LIN {X 0,Y 355.235,Z 349.049,A -85,B 0,C 180,E1 -13317.733,E2 -13317.733} C_VEL
LIN {X 0,Y 355.386,Z 349.032,A -85,B 0,C 180,E1 -13320.001,E2 -13320.001} C_VEL
LIN {X 0,Y 355.236,Z 349.048,A -85,B 0,C 180,E1 -13322.269,E2 -13322.269} C_VEL
LIN {X 0,Y 355.128,Z 349.059,A -85,B 0,C 180,E1 -13326.82,E2 -13326.82} C_VEL
LIN {X 0,Y 355.007,Z 349.075,A -85,B 0,C 180,E1 -13329.114,E2 -13329.114} C_VEL
LIN {X 0,Y 354.917,Z 349.085,A -85,B 0,C 180,E1 -13332.582,E2 -13332.582} C_VEL
LIN {X 0,Y 354.88,Z 349.091,A -85,B 0,C 180,E1 -13336.097,E2 -13336.097} C_VEL
LIN {X 0,Y 354.892,Z 349.088,A -85,B 0,C 180,E1 -13338.474,E2 -13338.474} C_VEL
LIN {X 0,Y 354.826,Z 349.097,A -85,B 0,C 180,E1 -13342.108,E2 -13342.108} C_VEL
LIN {X 0,Y 354.891,Z 349.09,A -85,B 0,C 180,E1 -13345.829,E2 -13345.829} C_VEL
LIN {X 0,Y 354.847,Z 349.096,A -85,B 0,C 180,E1 -13349.68,E2 -13349.68} C_VEL
LIN {X 0,Y 354.799,Z 349.101,A -85,B 0,C 180,E1 -13353.704,E2 -13353.704} C_VEL
LIN {X 0,Y 354.792,Z 349.102,A -85,B 0,C 180,E1 -13356.461,E2 -13356.461} C_VEL
LIN {X 0,Y 354.818,Z 349.099,A -85,B 0,C 180,E1 -13359.425,E2 -13359.425} C_VEL
LIN {X 0,Y 354.783,Z 349.107,A -85,B 0,C 180,E1 -13362.869,E2 -13362.869} C_VEL
LIN {X 0,Y 354.771,Z 349.104,A -85,B 0,C 180,E1 -13366.107,E2 -13366.107} C_VEL
LIN {X 0,Y 354.897,Z 349.091,A -85,B 0,C 180,E1 -13370.299,E2 -13370.299} C_VEL
LIN {X 0,Y 354.925,Z 349.475,A -85,B 0,C 180,E1 -13370.683,E2 -13370.683} C_VEL
LIN {X 0,Y 355.893,Z 355.008,A -85,B 0,C 180,E1 -13374.062,E2 -13374.062} C_VEL
LIN {X 0,Y 356.377,Z 359.185,A -85,B 0,C 180,E1 -13376.485,E2 -13376.485} C_VEL
LIN {X 0,Y 356.221,Z 361.976,A -85,B 0,C 180,E1 -13378.035,E2 -13378.035} C_VEL
LIN {X 0,Y 355.439,Z 368.762,A -85,B 0,C 180,E1 -13381.672,E2 -13381.672} C_VEL
LIN {X 0,Y 354.767,Z 375.912,A -85,B 0,C 180,E1 -13385.419,E2 -13385.419} C_VEL
LIN {X 0,Y 354.249,Z 383.077,A -85,B 0,C 180,E1 -13389.079,E2 -13389.079} C_VEL
LIN {X 0,Y 353.744,Z 391.414,A -85,B 0,C 180,E1 -13393.259,E2 -13393.259} C_VEL
LIN {X 0,Y 353.648,Z 393.722,A -85,B 0,C 180,E1 -13394.347,E2 -13394.347} C_VEL
LIN {X 0,Y 355.033,Z 405.955,A -85,B 0,C 180,E1 -13394.943,E2 -13394.943} C_VEL
LIN {X 0,Y 355.952,Z 415.878,A -85,B 0,C 180,E1 -13395.628,E2 -13395.628} C_VEL
LIN {X 0,Y 356.321,Z 423.872,A -85,B 0,C 180,E1 -13396.311,E2 -13396.311} C_VEL
LIN {X 0,Y 356.015,Z 430.965,A -85,B 0,C 180,E1 -13397.025,E2 -13397.025} C_VEL
LIN {X 0,Y 355.341,Z 439.04,A -85,B 0,C 180,E1 -13398.016,E2 -13398.016} C_VEL
LIN {X 0,Y 354.883,Z 444.875,A -85,B 0,C 180,E1 -13398.869,E2 -13398.869} C_VEL
LIN {X 0,Y 354.341,Z 451.371,A -85,B 0,C 180,E1 -13400.007,E2 -13400.007} C_VEL
LIN {X 0,Y 353.972,Z 456.779,A -85,B 0,C 180,E1 -13401.15,E2 -13401.15} C_VEL
LIN {X 0,Y 353.626,Z 462.253,A -85,B 0,C 180,E1 -13402.579,E2 -13402.579} C_VEL
LIN {X 0,Y 353.352,Z 466.492,A -85,B 0,C 180,E1 -13403.978,E2 -13403.978} C_VEL
LIN {X 0,Y 353.355,Z 469.884,A -85,B 0,C 180,E1 -13405.438,E2 -13405.438} C_VEL
LIN {X 0,Y 353.281,Z 471.864,A -85,B 0,C 180,E1 -13406.58,E2 -13406.58} C_VEL
LIN {X 0,Y 353.296,Z 473.328,A -85,B 0,C 180,E1 -13407.721,E2 -13407.721} C_VEL
LIN {X 0,Y 353.362,Z 474.262,A -85,B 0,C 180,E1 -13408.862,E2 -13408.862} C_VEL
LIN {X 0,Y 353.395,Z 474.597,A -85,B 0,C 180,E1 -13410.001,E2 -13410.001} C_VEL
LIN {X 0,Y 353.356,Z 474.442,A -85,B 0,C 180,E1 -13411.141,E2 -13411.141} C_VEL
LIN {X 0,Y 353.261,Z 473.814,A -85,B 0,C 180,E1 -13412.282,E2 -13412.282} C_VEL
LIN {X 0,Y 353.272,Z 472.711,A -85,B 0,C 180,E1 -13413.423,E2 -13413.423} C_VEL
LIN {X 0,Y 353.325,Z 469.93,A -85,B 0,C 180,E1 -13415.137,E2 -13415.137} C_VEL
LIN {X 0,Y 353.412,Z 467.446,A -85,B 0,C 180,E1 -13416.28,E2 -13416.28} C_VEL
LIN {X 0,Y 353.649,Z 464.318,A -85,B 0,C 180,E1 -13417.423,E2 -13417.423} C_VEL
LIN {X 0,Y 354.118,Z 458.219,A -85,B 0,C 180,E1 -13419.137,E2 -13419.137} C_VEL
LIN {X 0,Y 354.581,Z 453.195,A -85,B 0,C 180,E1 -13420.277,E2 -13420.277} C_VEL
LIN {X 0,Y 355.196,Z 447.164,A -85,B 0,C 180,E1 -13421.413,E2 -13421.413} C_VEL
LIN {X 0,Y 355.86,Z 439.855,A -85,B 0,C 180,E1 -13422.549,E2 -13422.549} C_VEL
LIN {X 0,Y 356.656,Z 432.1,A -85,B 0,C 180,E1 -13423.534,E2 -13423.534} C_VEL
LIN {X 0,Y 357.137,Z 425.476,A -85,B 0,C 180,E1 -13424.241,E2 -13424.241} C_VEL
LIN {X 0,Y 356.862,Z 416.272,A -85,B 0,C 180,E1 -13425.081,E2 -13425.081} C_VEL
LIN {X 0,Y 356.041,Z 407.363,A -85,B 0,C 180,E1 -13425.75,E2 -13425.75} C_VEL
LIN {X 0,Y 354.507,Z 396.758,A -85,B 0,C 180,E1 -13426.388,E2 -13426.388} C_VEL
LIN {X 0,Y 353.78,Z 392.415,A -85,B 0,C 180,E1 -13426.594,E2 -13426.594} C_VEL
LIN {X 0,Y 354.187,Z 385.023,A -85,B 0,C 180,E1 -13430.32,E2 -13430.32} C_VEL
LIN {X 0,Y 354.791,Z 377.309,A -85,B 0,C 180,E1 -13434.326,E2 -13434.326} C_VEL
LIN {X 0,Y 355.443,Z 371.062,A -85,B 0,C 180,E1 -13437.689,E2 -13437.689} C_VEL
LIN {X 0,Y 356.313,Z 364.375,A -85,B 0,C 180,E1 -13441.442,E2 -13441.442} C_VEL
LIN {X 0,Y 356.63,Z 360.91,A -85,B 0,C 180,E1 -13443.491,E2 -13443.491} C_VEL
LIN {X 0,Y 356.164,Z 356.993,A -85,B 0,C 180,E1 -13445.998,E2 -13445.998} C_VEL
LIN {X 0,Y 355.369,Z 351.925,A -85,B 0,C 180,E1 -13449.529,E2 -13449.529} C_VEL
LIN {X 0,Y 354.824,Z 349.11,A -85,B 0,C 180,E1 -13451.712,E2 -13451.712} C_VEL
LIN {X 0,Y 354.771,Z 349.112,A -85,B 0,C 180,E1 -13455.494,E2 -13455.494} C_VEL
LIN {X 0,Y 354.795,Z 349.105,A -85,B 0,C 180,E1 -13459.179,E2 -13459.179} C_VEL
LIN {X 0,Y 354.814,Z 349.102,A -85,B 0,C 180,E1 -13462.403,E2 -13462.403} C_VEL
LIN {X 0,Y 354.819,Z 349.102,A -85,B 0,C 180,E1 -13464.941,E2 -13464.941} C_VEL
LIN {X 0,Y 354.801,Z 349.103,A -85,B 0,C 180,E1 -13468.405,E2 -13468.405} C_VEL
LIN {X 0,Y 354.854,Z 349.097,A -85,B 0,C 180,E1 -13471.618,E2 -13471.618} C_VEL
LIN {X 0,Y 354.907,Z 349.091,A -85,B 0,C 180,E1 -13474.172,E2 -13474.172} C_VEL
LIN {X 0,Y 354.843,Z 349.098,A -85,B 0,C 180,E1 -13477.894,E2 -13477.894} C_VEL
LIN {X 0,Y 354.93,Z 349.087,A -85,B 0,C 180,E1 -13481.891,E2 -13481.891} C_VEL
LIN {X 0,Y 354.95,Z 349.085,A -85,B 0,C 180,E1 -13485.981,E2 -13485.981} C_VEL
LIN {X 0,Y 354.963,Z 349.084,A -85,B 0,C 180,E1 -13489.734,E2 -13489.734} C_VEL
LIN {X 0,Y 355.106,Z 349.065,A -85,B 0,C 180,E1 -13493.179,E2 -13493.179} C_VEL
LIN {X 0,Y 355.246,Z 349.048,A -85,B 0,C 180,E1 -13497.731,E2 -13497.731} C_VEL
LIN {X 0,Y 355.381,Z 349.033,A -85,B 0,C 180,E1 -13499.999,E2 -13499.999} C_VEL
LIN {X 0,Y 355.248,Z 349.048,A -85,B 0,C 180,E1 -13502.266,E2 -13502.266} C_VEL
LIN {X 0,Y 355.117,Z 349.065,A -85,B 0,C 180,E1 -13506.818,E2 -13506.818} C_VEL
LIN {X 0,Y 354.96,Z 349.084,A -85,B 0,C 180,E1 -13510.263,E2 -13510.263} C_VEL
LIN {X 0,Y 354.943,Z 349.089,A -85,B 0,C 180,E1 -13514.015,E2 -13514.015} C_VEL
LIN {X 0,Y 354.751,Z 349.114,A -85,B 0,C 180,E1 -13517.286,E2 -13517.286} C_VEL
LIN {X 0,Y 354.61,Z 349.14,A -85,B 0,C 180,E1 -13518.486,E2 -13518.486} C_VEL
LIN {X 0,Y 354.486,Z 351.743,A -85,B 0,C 180,E1 -13521.278,E2 -13521.278} C_VEL
LIN {X 0,Y 354.24,Z 354.97,A -85,B 0,C 180,E1 -13524.621,E2 -13524.621} C_VEL
LIN {X 0,Y 354.088,Z 357.477,A -85,B 0,C 180,E1 -13527.16,E2 -13527.16} C_VEL
LIN {X 0,Y 353.925,Z 360.115,A -85,B 0,C 180,E1 -13529.763,E2 -13529.763} C_VEL
LIN {X 0,Y 353.767,Z 363.986,A -85,B 0,C 180,E1 -13533.509,E2 -13533.509} C_VEL
LIN {X 0,Y 356.374,Z 374.506,A -85,B 0,C 180,E1 -13534.195,E2 -13534.195} C_VEL
LIN {X 0,Y 358.039,Z 383.016,A -85,B 0,C 180,E1 -13534.867,E2 -13534.867} C_VEL
LIN {X 0,Y 358.578,Z 389.237,A -85,B 0,C 180,E1 -13535.407,E2 -13535.407} C_VEL
LIN {X 0,Y 357.779,Z 399.313,A -85,B 0,C 180,E1 -13536.426,E2 -13536.426} C_VEL
LIN {X 0,Y 357.04,Z 406.286,A -85,B 0,C 180,E1 -13537.29,E2 -13537.29} C_VEL
LIN {X 0,Y 356.525,Z 412.401,A -85,B 0,C 180,E1 -13538.2,E2 -13538.2} C_VEL
LIN {X 0,Y 355.812,Z 419.035,A -85,B 0,C 180,E1 -13539.391,E2 -13539.391} C_VEL
LIN {X 0,Y 355.266,Z 423.977,A -85,B 0,C 180,E1 -13540.454,E2 -13540.454} C_VEL
LIN {X 0,Y 354.667,Z 429.227,A -85,B 0,C 180,E1 -13541.838,E2 -13541.838} C_VEL
LIN {X 0,Y 354.332,Z 432.253,A -85,B 0,C 180,E1 -13542.786,E2 -13542.786} C_VEL
LIN {X 0,Y 353.898,Z 436.127,A -85,B 0,C 180,E1 -13544.362,E2 -13544.362} C_VEL
LIN {X 0,Y 353.594,Z 438.873,A -85,B 0,C 180,E1 -13545.919,E2 -13545.919} C_VEL
LIN {X 0,Y 353.3,Z 440.605,A -85,B 0,C 180,E1 -13547.44,E2 -13547.44} C_VEL
LIN {X 0,Y 353.163,Z 441.468,A -85,B 0,C 180,E1 -13549.128,E2 -13549.128} C_VEL
LIN {X 0,Y 353.164,Z 441.225,A -85,B 0,C 180,E1 -13550.903,E2 -13550.903} C_VEL
LIN {X 0,Y 353.286,Z 439.695,A -85,B 0,C 180,E1 -13552.721,E2 -13552.721} C_VEL
LIN {X 0,Y 353.468,Z 437.782,A -85,B 0,C 180,E1 -13554.02,E2 -13554.02} C_VEL
LIN {X 0,Y 353.702,Z 434.686,A -85,B 0,C 180,E1 -13555.507,E2 -13555.507} C_VEL
LIN {X 0,Y 354.067,Z 430.281,A -85,B 0,C 180,E1 -13557.061,E2 -13557.061} C_VEL
LIN {X 0,Y 354.468,Z 425.095,A -85,B 0,C 180,E1 -13558.488,E2 -13558.488} C_VEL
LIN {X 0,Y 354.94,Z 419.788,A -85,B 0,C 180,E1 -13559.673,E2 -13559.673} C_VEL
LIN {X 0,Y 355.448,Z 413.918,A -85,B 0,C 180,E1 -13560.762,E2 -13560.762} C_VEL
LIN {X 0,Y 355.894,Z 407.866,A -85,B 0,C 180,E1 -13561.708,E2 -13561.708} C_VEL
LIN {X 0,Y 356.453,Z 400.719,A -85,B 0,C 180,E1 -13562.641,E2 -13562.641} C_VEL
LIN {X 0,Y 357.061,Z 392.116,A -85,B 0,C 180,E1 -13563.555,E2 -13563.555} C_VEL
LIN {X 0,Y 357.398,Z 384.562,A -85,B 0,C 180,E1 -13564.209,E2 -13564.209} C_VEL
LIN {X 0,Y 356.037,Z 375.647,A -85,B 0,C 180,E1 -13564.886,E2 -13564.886} C_VEL
LIN {X 0,Y 354.144,Z 365.686,A -85,B 0,C 180,E1 -13565.481,E2 -13565.481} C_VEL
LIN {X 0,Y 353.599,Z 362.774,A -85,B 0,C 180,E1 -13565.663,E2 -13565.663} C_VEL
LIN {X 0,Y 353.651,Z 358.953,A -85,B 0,C 180,E1 -13569.065,E2 -13569.065} C_VEL
LIN {X 0,Y 353.885,Z 354.967,A -85,B 0,C 180,E1 -13572.668,E2 -13572.668} C_VEL
LIN {X 0,Y 354.106,Z 350.778,A -85,B 0,C 180,E1 -13576.527,E2 -13576.527} C_VEL
LIN {X 0,Y 354.133,Z 349.869,A -85,B 0,C 180,E1 -13577.389,E2 -13577.389} C_VEL
LIN {X 0,Y 354.239,Z 349.175,A -85,B 0,C 180,E1 -13578.555,E2 -13578.555} C_VEL
LIN {X 0,Y 354.905,Z 349.09,A -85,B 0,C 180,E1 -13582.031,E2 -13582.031} C_VEL
LIN {X 0,Y 355.06,Z 349.072,A -85,B 0,C 180,E1 -13584.319,E2 -13584.319} C_VEL
LIN {X 0,Y 355.236,Z 349.047,A -85,B 0,C 180,E1 -13587.731,E2 -13587.731} C_VEL
LIN {X 0,Y 355.387,Z 349.031,A -85,B 0,C 180,E1 -13589.999,E2 -13589.999} C_VEL
LIN {X 0,Y 355.236,Z 349.049,A -85,B 0,C 180,E1 -13592.266,E2 -13592.266} C_VEL
LIN {X 0,Y 355.131,Z 349.059,A -85,B 0,C 180,E1 -13596.818,E2 -13596.818} C_VEL
LIN {X 0,Y 355.005,Z 349.074,A -85,B 0,C 180,E1 -13599.111,E2 -13599.111} C_VEL
LIN {X 0,Y 354.914,Z 349.086,A -85,B 0,C 180,E1 -13602.579,E2 -13602.579} C_VEL
LIN {X 0,Y 354.877,Z 349.093,A -85,B 0,C 180,E1 -13606.095,E2 -13606.095} C_VEL
LIN {X 0,Y 354.888,Z 349.089,A -85,B 0,C 180,E1 -13608.471,E2 -13608.471} C_VEL
LIN {X 0,Y 354.821,Z 349.099,A -85,B 0,C 180,E1 -13612.105,E2 -13612.105} C_VEL
LIN {X 0,Y 354.886,Z 349.092,A -85,B 0,C 180,E1 -13615.827,E2 -13615.827} C_VEL
LIN {X 0,Y 354.84,Z 349.098,A -85,B 0,C 180,E1 -13619.678,E2 -13619.678} C_VEL
LIN {X 0,Y 354.792,Z 349.103,A -85,B 0,C 180,E1 -13623.701,E2 -13623.701} C_VEL
LIN {X 0,Y 354.789,Z 349.101,A -85,B 0,C 180,E1 -13626.458,E2 -13626.458} C_VEL
LIN {X 0,Y 354.811,Z 349.102,A -85,B 0,C 180,E1 -13629.424,E2 -13629.424} C_VEL
LIN {X 0,Y 354.827,Z 349.1,A -85,B 0,C 180,E1 -13632.876,E2 -13632.876} C_VEL
LIN {X 0,Y 354.853,Z 349.093,A -85,B 0,C 180,E1 -13634.072,E2 -13634.072} C_VEL
LIN {X 0,Y 354.196,Z 349.18,A -85,B 0,C 180,E1 -13635.018,E2 -13635.018} C_VEL
LIN {X 0,Y 351.315,Z 349.536,A -85,B 0,C 180,E1 -13636.556,E2 -13636.556} C_VEL
LIN {X 0,Y 348.871,Z 349.838,A -85,B 0,C 180,E1 -13637.801,E2 -13637.801} C_VEL
LIN {X 0,Y 347.831,Z 349.972,A -85,B 0,C 180,E1 -13638.765,E2 -13638.765} C_VEL
LIN {X 0,Y 347.752,Z 349.975,A -85,B 0,C 180,E1 -13639.092,E2 -13639.092} C_VEL
LIN {X 0,Y 347.752,Z 349.982,A -85,B 0,C 180,E1 -13642.68,E2 -13642.68} C_VEL
LIN {X 0,Y 347.734,Z 349.98,A -85,B 0,C 180,E1 -13645.956,E2 -13645.956} C_VEL
LIN {X 0,Y 347.75,Z 349.978,A -85,B 0,C 180,E1 -13649.654,E2 -13649.654} C_VEL
LIN {X 0,Y 347.838,Z 349.971,A -85,B 0,C 180,E1 -13652.745,E2 -13652.745} C_VEL
LIN {X 0,Y 347.804,Z 349.974,A -85,B 0,C 180,E1 -13656.165,E2 -13656.165} C_VEL
LIN {X 0,Y 347.83,Z 349.969,A -85,B 0,C 180,E1 -13659.912,E2 -13659.912} C_VEL
LIN {X 0,Y 347.854,Z 349.97,A -85,B 0,C 180,E1 -13662.36,E2 -13662.36} C_VEL
LIN {X 0,Y 347.884,Z 349.964,A -85,B 0,C 180,E1 -13665.972,E2 -13665.972} C_VEL
LIN {X 0,Y 347.92,Z 349.957,A -85,B 0,C 180,E1 -13669.527,E2 -13669.527} C_VEL
LIN {X 0,Y 348.062,Z 349.942,A -85,B 0,C 180,E1 -13671.876,E2 -13671.876} C_VEL
LIN {X 0,Y 348.056,Z 349.944,A -85,B 0,C 180,E1 -13674.207,E2 -13674.207} C_VEL
LIN {X 0,Y 348.197,Z 349.925,A -85,B 0,C 180,E1 -13677.688,E2 -13677.688} C_VEL
LIN {X 0,Y 348.335,Z 349.91,A -85,B 0,C 180,E1 -13680.001,E2 -13680.001} C_VEL
LIN {X 0,Y 348.199,Z 349.924,A -85,B 0,C 180,E1 -13682.315,E2 -13682.315} C_VEL
LIN {X 0,Y 348.096,Z 349.935,A -85,B 0,C 180,E1 -13686.959,E2 -13686.959} C_VEL
LIN {X 0,Y 347.959,Z 349.954,A -85,B 0,C 180,E1 -13689.3,E2 -13689.3} C_VEL
LIN {X 0,Y 347.884,Z 349.961,A -85,B 0,C 180,E1 -13692.841,E2 -13692.841} C_VEL
LIN {X 0,Y 347.83,Z 349.968,A -85,B 0,C 180,E1 -13696.433,E2 -13696.433} C_VEL
LIN {X 0,Y 347.842,Z 349.967,A -85,B 0,C 180,E1 -13698.862,E2 -13698.862} C_VEL
LIN {X 0,Y 347.766,Z 349.976,A -85,B 0,C 180,E1 -13702.581,E2 -13702.581} C_VEL
LIN {X 0,Y 347.805,Z 349.974,A -85,B 0,C 180,E1 -13705.11,E2 -13705.11} C_VEL
LIN {X 0,Y 347.805,Z 349.973,A -85,B 0,C 180,E1 -13707.695,E2 -13707.695} C_VEL
LIN {X 0,Y 347.757,Z 349.977,A -85,B 0,C 180,E1 -13710.348,E2 -13710.348} C_VEL
LIN {X 0,Y 347.738,Z 349.98,A -85,B 0,C 180,E1 -13714.466,E2 -13714.466} C_VEL
LIN {X 0,Y 347.768,Z 349.976,A -85,B 0,C 180,E1 -13717.991,E2 -13717.991} C_VEL
LIN {X 0,Y 347.745,Z 349.979,A -85,B 0,C 180,E1 -13721.832,E2 -13721.832} C_VEL
LIN {X 0,Y 347.762,Z 349.981,A -85,B 0,C 180,E1 -13725.019,E2 -13725.019} C_VEL
LIN {X 0,Y 347.746,Z 349.981,A -85,B 0,C 180,E1 -13728.399,E2 -13728.399} C_VEL
LIN {X 0,Y 347.86,Z 349.982,A -85,B 0,C 180,E1 -13730.252,E2 -13730.252} C_VEL
LIN {X 0,Y 348.952,Z 356.424,A -85,B 0,C 180,E1 -13734.265,E2 -13734.265} C_VEL
LIN {X 0,Y 349.359,Z 360.053,A -85,B 0,C 180,E1 -13736.414,E2 -13736.414} C_VEL
LIN {X 0,Y 349.058,Z 363.639,A -85,B 0,C 180,E1 -13738.435,E2 -13738.435} C_VEL
LIN {X 0,Y 348.247,Z 370.795,A -85,B 0,C 180,E1 -13742.346,E2 -13742.346} C_VEL
LIN {X 0,Y 347.562,Z 377.946,A -85,B 0,C 180,E1 -13746.147,E2 -13746.147} C_VEL
LIN {X 0,Y 347.117,Z 383.903,A -85,B 0,C 180,E1 -13749.25,E2 -13749.25} C_VEL
LIN {X 0,Y 346.637,Z 392.186,A -85,B 0,C 180,E1 -13753.512,E2 -13753.512} C_VEL
LIN {X 0,Y 346.565,Z 393.22,A -85,B 0,C 180,E1 -13754.038,E2 -13754.038} C_VEL
LIN {X 0,Y 348.011,Z 406.017,A -85,B 0,C 180,E1 -13754.706,E2 -13754.706} C_VEL
LIN {X 0,Y 348.936,Z 416.263,A -85,B 0,C 180,E1 -13755.44,E2 -13755.44} C_VEL
LIN {X 0,Y 349.314,Z 424.538,A -85,B 0,C 180,E1 -13756.179,E2 -13756.179} C_VEL
LIN {X 0,Y 348.983,Z 431.452,A -85,B 0,C 180,E1 -13756.907,E2 -13756.907} C_VEL
LIN {X 0,Y 348.289,Z 439.389,A -85,B 0,C 180,E1 -13757.917,E2 -13757.917} C_VEL
LIN {X 0,Y 347.758,Z 445.969,A -85,B 0,C 180,E1 -13758.933,E2 -13758.933} C_VEL
LIN {X 0,Y 347.2,Z 452.227,A -85,B 0,C 180,E1 -13760.094,E2 -13760.094} C_VEL
LIN {X 0,Y 346.851,Z 457.431,A -85,B 0,C 180,E1 -13761.261,E2 -13761.261} C_VEL
LIN {X 0,Y 346.552,Z 461.761,A -85,B 0,C 180,E1 -13762.427,E2 -13762.427} C_VEL
LIN {X 0,Y 346.25,Z 466.876,A -85,B 0,C 180,E1 -13764.177,E2 -13764.177} C_VEL
LIN {X 0,Y 346.235,Z 470.601,A -85,B 0,C 180,E1 -13765.928,E2 -13765.928} C_VEL
LIN {X 0,Y 346.199,Z 472.955,A -85,B 0,C 180,E1 -13767.675,E2 -13767.675} C_VEL
LIN {X 0,Y 346.267,Z 473.896,A -85,B 0,C 180,E1 -13768.839,E2 -13768.839} C_VEL
LIN {X 0,Y 346.316,Z 474.249,A -85,B 0,C 180,E1 -13770.001,E2 -13770.001} C_VEL
LIN {X 0,Y 346.258,Z 474.118,A -85,B 0,C 180,E1 -13771.164,E2 -13771.164} C_VEL
LIN {X 0,Y 346.167,Z 473.514,A -85,B 0,C 180,E1 -13772.329,E2 -13772.329} C_VEL
LIN {X 0,Y 346.196,Z 472.431,A -85,B 0,C 180,E1 -13773.493,E2 -13773.493} C_VEL
LIN {X 0,Y 346.225,Z 469.677,A -85,B 0,C 180,E1 -13775.242,E2 -13775.242} C_VEL
LIN {X 0,Y 346.349,Z 467.218,A -85,B 0,C 180,E1 -13776.409,E2 -13776.409} C_VEL
LIN {X 0,Y 346.731,Z 462.216,A -85,B 0,C 180,E1 -13778.158,E2 -13778.158} C_VEL
LIN {X 0,Y 347.206,Z 456.876,A -85,B 0,C 180,E1 -13779.614,E2 -13779.614} C_VEL
LIN {X 0,Y 347.728,Z 451.66,A -85,B 0,C 180,E1 -13780.776,E2 -13780.776} C_VEL
LIN {X 0,Y 348.397,Z 445.409,A -85,B 0,C 180,E1 -13781.934,E2 -13781.934} C_VEL
LIN {X 0,Y 349.066,Z 438.865,A -85,B 0,C 180,E1 -13782.945,E2 -13782.945} C_VEL
LIN {X 0,Y 349.899,Z 430.982,A -85,B 0,C 180,E1 -13783.949,E2 -13783.949} C_VEL
LIN {X 0,Y 350.203,Z 424.211,A -85,B 0,C 180,E1 -13784.677,E2 -13784.677} C_VEL
LIN {X 0,Y 349.949,Z 416.162,A -85,B 0,C 180,E1 -13785.423,E2 -13785.423} C_VEL
LIN {X 0,Y 349.041,Z 406.753,A -85,B 0,C 180,E1 -13786.149,E2 -13786.149} C_VEL
LIN {X 0,Y 347.447,Z 396.284,A -85,B 0,C 180,E1 -13786.797,E2 -13786.797} C_VEL
LIN {X 0,Y 346.726,Z 392.047,A -85,B 0,C 180,E1 -13787.018,E2 -13787.018} C_VEL
LIN {X 0,Y 347.196,Z 384.835,A -85,B 0,C 180,E1 -13790.748,E2 -13790.748} C_VEL
LIN {X 0,Y 347.877,Z 376.673,A -85,B 0,C 180,E1 -13795.105,E2 -13795.105} C_VEL
LIN {X 0,Y 348.654,Z 369.825,A -85,B 0,C 180,E1 -13798.934,E2 -13798.934} C_VEL
LIN {X 0,Y 349.496,Z 363.911,A -85,B 0,C 180,E1 -13802.372,E2 -13802.372} C_VEL
LIN {X 0,Y 349.564,Z 360.528,A -85,B 0,C 180,E1 -13804.481,E2 -13804.481} C_VEL
LIN {X 0,Y 348.686,Z 355.14,A -85,B 0,C 180,E1 -13808.179,E2 -13808.179} C_VEL
LIN {X 0,Y 348.25,Z 352.379,A -85,B 0,C 180,E1 -13810.226,E2 -13810.226} C_VEL
LIN {X 0,Y 347.775,Z 349.987,A -85,B 0,C 180,E1 -13812.218,E2 -13812.218} C_VEL
LIN {X 0,Y 347.713,Z 349.992,A -85,B 0,C 180,E1 -13815.027,E2 -13815.027} C_VEL
LIN {X 0,Y 347.758,Z 349.982,A -85,B 0,C 180,E1 -13818.398,E2 -13818.398} C_VEL
LIN {X 0,Y 347.78,Z 349.978,A -85,B 0,C 180,E1 -13822.012,E2 -13822.012} C_VEL
LIN {X 0,Y 347.752,Z 349.982,A -85,B 0,C 180,E1 -13825.536,E2 -13825.536} C_VEL
LIN {X 0,Y 347.753,Z 349.981,A -85,B 0,C 180,E1 -13828.3,E2 -13828.3} C_VEL
LIN {X 0,Y 347.787,Z 349.976,A -85,B 0,C 180,E1 -13830.987,E2 -13830.987} C_VEL
LIN {X 0,Y 347.839,Z 349.97,A -85,B 0,C 180,E1 -13833.607,E2 -13833.607} C_VEL
LIN {X 0,Y 347.797,Z 349.976,A -85,B 0,C 180,E1 -13836.162,E2 -13836.162} C_VEL
LIN {X 0,Y 347.82,Z 349.973,A -85,B 0,C 180,E1 -13839.909,E2 -13839.909} C_VEL
LIN {X 0,Y 347.874,Z 349.967,A -85,B 0,C 180,E1 -13842.359,E2 -13842.359} C_VEL
LIN {X 0,Y 347.905,Z 349.962,A -85,B 0,C 180,E1 -13845.97,E2 -13845.97} C_VEL
LIN {X 0,Y 347.903,Z 349.963,A -85,B 0,C 180,E1 -13849.524,E2 -13849.524} C_VEL
LIN {X 0,Y 348.074,Z 349.942,A -85,B 0,C 180,E1 -13853.041,E2 -13853.041} C_VEL
LIN {X 0,Y 348.208,Z 349.925,A -85,B 0,C 180,E1 -13857.685,E2 -13857.685} C_VEL
LIN {X 0,Y 348.331,Z 349.911,A -85,B 0,C 180,E1 -13859.999,E2 -13859.999} C_VEL
LIN {X 0,Y 348.211,Z 349.925,A -85,B 0,C 180,E1 -13862.312,E2 -13862.312} C_VEL
LIN {X 0,Y 348.083,Z 349.941,A -85,B 0,C 180,E1 -13866.957,E2 -13866.957} C_VEL
LIN {X 0,Y 347.901,Z 349.963,A -85,B 0,C 180,E1 -13870.474,E2 -13870.474} C_VEL
LIN {X 0,Y 347.903,Z 349.966,A -85,B 0,C 180,E1 -13874.148,E2 -13874.148} C_VEL
LIN {X 0,Y 347.683,Z 349.994,A -85,B 0,C 180,E1 -13877.649,E2 -13877.649} C_VEL
LIN {X 0,Y 347.61,Z 350.001,A -85,B 0,C 180,E1 -13878.146,E2 -13878.146} C_VEL
LIN {X 0,Y 347.448,Z 352.93,A -85,B 0,C 180,E1 -13881.49,E2 -13881.49} C_VEL
LIN {X 0,Y 347.153,Z 356.419,A -85,B 0,C 180,E1 -13885.158,E2 -13885.158} C_VEL
LIN {X 0,Y 346.966,Z 360.281,A -85,B 0,C 180,E1 -13889.085,E2 -13889.085} C_VEL
LIN {X 0,Y 346.725,Z 364.356,A -85,B 0,C 180,E1 -13893.092,E2 -13893.092} C_VEL
LIN {X 0,Y 349.503,Z 375.389,A -85,B 0,C 180,E1 -13893.853,E2 -13893.853} C_VEL
LIN {X 0,Y 351.333,Z 384.787,A -85,B 0,C 180,E1 -13894.634,E2 -13894.634} C_VEL
LIN {X 0,Y 351.797,Z 389.821,A -85,B 0,C 180,E1 -13895.087,E2 -13895.087} C_VEL
LIN {X 0,Y 351.016,Z 399.003,A -85,B 0,C 180,E1 -13896.023,E2 -13896.023} C_VEL
LIN {X 0,Y 350.178,Z 406.881,A -85,B 0,C 180,E1 -13897.018,E2 -13897.018} C_VEL
LIN {X 0,Y 349.563,Z 413.623,A -85,B 0,C 180,E1 -13898.061,E2 -13898.061} C_VEL
LIN {X 0,Y 348.812,Z 420.123,A -85,B 0,C 180,E1 -13899.277,E2 -13899.277} C_VEL
LIN {X 0,Y 348.166,Z 425.721,A -85,B 0,C 180,E1 -13900.558,E2 -13900.558} C_VEL
LIN {X 0,Y 347.581,Z 430.333,A -85,B 0,C 180,E1 -13901.853,E2 -13901.853} C_VEL
LIN {X 0,Y 347.139,Z 434.19,A -85,B 0,C 180,E1 -13903.209,E2 -13903.209} C_VEL
LIN {X 0,Y 346.646,Z 438.389,A -85,B 0,C 180,E1 -13905.2,E2 -13905.2} C_VEL
LIN {X 0,Y 346.301,Z 440.621,A -85,B 0,C 180,E1 -13906.934,E2 -13906.934} C_VEL
LIN {X 0,Y 346.104,Z 441.717,A -85,B 0,C 180,E1 -13908.703,E2 -13908.703} C_VEL
LIN {X 0,Y 346.066,Z 441.902,A -85,B 0,C 180,E1 -13909.467,E2 -13909.467} C_VEL
LIN {X 0,Y 346.078,Z 441.527,A -85,B 0,C 180,E1 -13910.983,E2 -13910.983} C_VEL
LIN {X 0,Y 346.179,Z 440.317,A -85,B 0,C 180,E1 -13912.478,E2 -13912.478} C_VEL
LIN {X 0,Y 346.405,Z 437.763,A -85,B 0,C 180,E1 -13914.243,E2 -13914.243} C_VEL
LIN {X 0,Y 346.67,Z 434.306,A -85,B 0,C 180,E1 -13915.843,E2 -13915.843} C_VEL
LIN {X 0,Y 347.024,Z 430.479,A -85,B 0,C 180,E1 -13917.196,E2 -13917.196} C_VEL
LIN {X 0,Y 347.441,Z 425.439,A -85,B 0,C 180,E1 -13918.608,E2 -13918.608} C_VEL
LIN {X 0,Y 347.852,Z 420.906,A -85,B 0,C 180,E1 -13919.661,E2 -13919.661} C_VEL
LIN {X 0,Y 348.355,Z 415.248,A -85,B 0,C 180,E1 -13920.762,E2 -13920.762} C_VEL
LIN {X 0,Y 348.923,Z 408.14,A -85,B 0,C 180,E1 -13921.904,E2 -13921.904} C_VEL
LIN {X 0,Y 349.553,Z 400.25,A -85,B 0,C 180,E1 -13922.941,E2 -13922.941} C_VEL
LIN {X 0,Y 350.131,Z 392.298,A -85,B 0,C 180,E1 -13923.793,E2 -13923.793} C_VEL
LIN {X 0,Y 350.375,Z 384.864,A -85,B 0,C 180,E1 -13924.452,E2 -13924.452} C_VEL
LIN {X 0,Y 349.013,Z 376.145,A -85,B 0,C 180,E1 -13925.132,E2 -13925.132} C_VEL
LIN {X 0,Y 347.235,Z 366.83,A -85,B 0,C 180,E1 -13925.709,E2 -13925.709} C_VEL
LIN {X 0,Y 346.52,Z 363.103,A -85,B 0,C 180,E1 -13925.917,E2 -13925.917} C_VEL
LIN {X 0,Y 346.602,Z 358.767,A -85,B 0,C 180,E1 -13929.835,E2 -13929.835} C_VEL
LIN {X 0,Y 346.807,Z 356.093,A -85,B 0,C 180,E1 -13932.302,E2 -13932.302} C_VEL
LIN {X 0,Y 347.034,Z 351.663,A -85,B 0,C 180,E1 -13936.421,E2 -13936.421} C_VEL
LIN {X 0,Y 347.142,Z 350.059,A -85,B 0,C 180,E1 -13938.318,E2 -13938.318} C_VEL
LIN {X 0,Y 347.858,Z 349.966,A -85,B 0,C 180,E1 -13941.868,E2 -13941.868} C_VEL
LIN {X 0,Y 348.03,Z 349.948,A -85,B 0,C 180,E1 -13944.204,E2 -13944.204} C_VEL
LIN {X 0,Y 348.198,Z 349.924,A -85,B 0,C 180,E1 -13947.685,E2 -13947.685} C_VEL
LIN {X 0,Y 348.336,Z 349.909,A -85,B 0,C 180,E1 -13949.999,E2 -13949.999} C_VEL
LIN {X 0,Y 348.199,Z 349.926,A -85,B 0,C 180,E1 -13952.312,E2 -13952.312} C_VEL
LIN {X 0,Y 348.099,Z 349.934,A -85,B 0,C 180,E1 -13956.956,E2 -13956.956} C_VEL
LIN {X 0,Y 347.958,Z 349.953,A -85,B 0,C 180,E1 -13959.297,E2 -13959.297} C_VEL
LIN {X 0,Y 347.882,Z 349.961,A -85,B 0,C 180,E1 -13962.838,E2 -13962.838} C_VEL
LIN {X 0,Y 347.827,Z 349.969,A -85,B 0,C 180,E1 -13966.43,E2 -13966.43} C_VEL
LIN {X 0,Y 347.838,Z 349.967,A -85,B 0,C 180,E1 -13968.859,E2 -13968.859} C_VEL
LIN {X 0,Y 347.761,Z 349.976,A -85,B 0,C 180,E1 -13972.578,E2 -13972.578} C_VEL
LIN {X 0,Y 347.799,Z 349.974,A -85,B 0,C 180,E1 -13975.108,E2 -13975.108} C_VEL
LIN {X 0,Y 347.799,Z 349.975,A -85,B 0,C 180,E1 -13977.693,E2 -13977.693} C_VEL
LIN {X 0,Y 347.75,Z 349.978,A -85,B 0,C 180,E1 -13980.346,E2 -13980.346} C_VEL
LIN {X 0,Y 347.73,Z 349.98,A -85,B 0,C 180,E1 -13984.463,E2 -13984.463} C_VEL
LIN {X 0,Y 347.767,Z 349.976,A -85,B 0,C 180,E1 -13987.99,E2 -13987.99} C_VEL
LIN {X 0,Y 347.769,Z 349.976,A -85,B 0,C 180,E1 -13991.825,E2 -13991.825} C_VEL
LIN {X 0,Y 347.816,Z 349.975,A -85,B 0,C 180,E1 -13995.006,E2 -13995.006} C_VEL
LIN {X 0,Y 347.77,Z 349.976,A -85,B 0,C 180,E1 -13998.391,E2 -13998.391} C_VEL
LIN {X 0,Y 347.752,Z 349.975,A -85,B 0,C 180,E1 -13999.092,E2 -13999.092} C_VEL
LIN {X 0,Y 347.093,Z 350.06,A -85,B 0,C 180,E1 -14000.058,E2 -14000.058} C_VEL
LIN {X 0,Y 344.225,Z 350.417,A -85,B 0,C 180,E1 -14001.628,E2 -14001.628} C_VEL
LIN {X 0,Y 341.794,Z 350.725,A -85,B 0,C 180,E1 -14002.9,E2 -14002.9} C_VEL
LIN {X 0,Y 340.762,Z 350.849,A -85,B 0,C 180,E1 -14003.884,E2 -14003.884} C_VEL
LIN {X 0,Y 340.684,Z 350.859,A -85,B 0,C 180,E1 -14004.217,E2 -14004.217} C_VEL
LIN {X 0,Y 340.676,Z 350.859,A -85,B 0,C 180,E1 -14007.755,E2 -14007.755} C_VEL
LIN {X 0,Y 340.761,Z 350.851,A -85,B 0,C 180,E1 -14010.333,E2 -14010.333} C_VEL
LIN {X 0,Y 340.791,Z 350.846,A -85,B 0,C 180,E1 -14013.021,E2 -14013.021} C_VEL
LIN {X 0,Y 340.763,Z 350.85,A -85,B 0,C 180,E1 -14016.931,E2 -14016.931} C_VEL
LIN {X 0,Y 340.793,Z 350.847,A -85,B 0,C 180,E1 -14020.735,E2 -14020.735} C_VEL
LIN {X 0,Y 340.775,Z 350.847,A -85,B 0,C 180,E1 -14023.219,E2 -14023.219} C_VEL
LIN {X 0,Y 340.834,Z 350.84,A -85,B 0,C 180,E1 -14026.891,E2 -14026.891} C_VEL
LIN {X 0,Y 340.918,Z 350.832,A -85,B 0,C 180,E1 -14030.509,E2 -14030.509} C_VEL
LIN {X 0,Y 341.064,Z 350.811,A -85,B 0,C 180,E1 -14032.899,E2 -14032.899} C_VEL
LIN {X 0,Y 341.159,Z 350.801,A -85,B 0,C 180,E1 -14037.64,E2 -14037.64} C_VEL
LIN {X 0,Y 341.285,Z 350.788,A -85,B 0,C 180,E1 -14040.001,E2 -14040.001} C_VEL
LIN {X 0,Y 341.161,Z 350.8,A -85,B 0,C 180,E1 -14042.362,E2 -14042.362} C_VEL
LIN {X 0,Y 341.065,Z 350.811,A -85,B 0,C 180,E1 -14047.103,E2 -14047.103} C_VEL
LIN {X 0,Y 340.865,Z 350.835,A -85,B 0,C 180,E1 -14050.695,E2 -14050.695} C_VEL
LIN {X 0,Y 340.853,Z 350.837,A -85,B 0,C 180,E1 -14054.326,E2 -14054.326} C_VEL
LIN {X 0,Y 340.828,Z 350.84,A -85,B 0,C 180,E1 -14058.468,E2 -14058.468} C_VEL
LIN {X 0,Y 340.745,Z 350.852,A -85,B 0,C 180,E1 -14061.858,E2 -14061.858} C_VEL
LIN {X 0,Y 340.765,Z 350.851,A -85,B 0,C 180,E1 -14065.666,E2 -14065.666} C_VEL
LIN {X 0,Y 340.735,Z 350.851,A -85,B 0,C 180,E1 -14068.321,E2 -14068.321} C_VEL
LIN {X 0,Y 340.697,Z 350.86,A -85,B 0,C 180,E1 -14071.046,E2 -14071.046} C_VEL
LIN {X 0,Y 340.712,Z 350.859,A -85,B 0,C 180,E1 -14075.281,E2 -14075.281} C_VEL
LIN {X 0,Y 340.704,Z 350.856,A -85,B 0,C 180,E1 -14078.388,E2 -14078.388} C_VEL
LIN {X 0,Y 340.694,Z 350.857,A -85,B 0,C 180,E1 -14082.047,E2 -14082.047} C_VEL
LIN {X 0,Y 340.678,Z 350.859,A -85,B 0,C 180,E1 -14085.463,E2 -14085.463} C_VEL
LIN {X 0,Y 340.698,Z 350.861,A -85,B 0,C 180,E1 -14088.695,E2 -14088.695} C_VEL
LIN {X 0,Y 340.821,Z 351.016,A -85,B 0,C 180,E1 -14090.138,E2 -14090.138} C_VEL
LIN {X 0,Y 341.702,Z 356.085,A -85,B 0,C 180,E1 -14093.385,E2 -14093.385} C_VEL
LIN {X 0,Y 342.347,Z 360.924,A -85,B 0,C 180,E1 -14096.341,E2 -14096.341} C_VEL
LIN {X 0,Y 341.903,Z 365.688,A -85,B 0,C 180,E1 -14099.079,E2 -14099.079} C_VEL
LIN {X 0,Y 341.046,Z 372.837,A -85,B 0,C 180,E1 -14103.043,E2 -14103.043} C_VEL
LIN {X 0,Y 340.364,Z 379.95,A -85,B 0,C 180,E1 -14106.903,E2 -14106.903} C_VEL
LIN {X 0,Y 339.9,Z 385.867,A -85,B 0,C 180,E1 -14110.054,E2 -14110.054} C_VEL
LIN {X 0,Y 339.525,Z 392.975,A -85,B 0,C 180,E1 -14113.775,E2 -14113.775} C_VEL
LIN {X 0,Y 340.992,Z 406.026,A -85,B 0,C 180,E1 -14114.46,E2 -14114.46} C_VEL
LIN {X 0,Y 341.806,Z 414.96,A -85,B 0,C 180,E1 -14115.104,E2 -14115.104} C_VEL
LIN {X 0,Y 342.293,Z 423.698,A -85,B 0,C 180,E1 -14115.89,E2 -14115.89} C_VEL
LIN {X 0,Y 342.037,Z 430.711,A -85,B 0,C 180,E1 -14116.636,E2 -14116.636} C_VEL
LIN {X 0,Y 341.324,Z 438.717,A -85,B 0,C 180,E1 -14117.667,E2 -14117.667} C_VEL
LIN {X 0,Y 340.749,Z 445.351,A -85,B 0,C 180,E1 -14118.702,E2 -14118.702} C_VEL
LIN {X 0,Y 340.188,Z 451.658,A -85,B 0,C 180,E1 -14119.888,E2 -14119.888} C_VEL
LIN {X 0,Y 339.805,Z 456.903,A -85,B 0,C 180,E1 -14121.078,E2 -14121.078} C_VEL
LIN {X 0,Y 339.506,Z 461.27,A -85,B 0,C 180,E1 -14122.269,E2 -14122.269} C_VEL
LIN {X 0,Y 339.171,Z 466.417,A -85,B 0,C 180,E1 -14124.055,E2 -14124.055} C_VEL
LIN {X 0,Y 339.169,Z 470.181,A -85,B 0,C 180,E1 -14125.843,E2 -14125.843} C_VEL
LIN {X 0,Y 339.107,Z 472.581,A -85,B 0,C 180,E1 -14127.626,E2 -14127.626} C_VEL
LIN {X 0,Y 339.171,Z 473.527,A -85,B 0,C 180,E1 -14128.814,E2 -14128.814} C_VEL
LIN {X 0,Y 339.224,Z 473.9,A -85,B 0,C 180,E1 -14130.002,E2 -14130.002} C_VEL
LIN {X 0,Y 339.16,Z 473.793,A -85,B 0,C 180,E1 -14131.189,E2 -14131.189} C_VEL
LIN {X 0,Y 339.077,Z 473.216,A -85,B 0,C 180,E1 -14132.377,E2 -14132.377} C_VEL
LIN {X 0,Y 339.121,Z 472.152,A -85,B 0,C 180,E1 -14133.566,E2 -14133.566} C_VEL
LIN {X 0,Y 339.133,Z 469.151,A -85,B 0,C 180,E1 -14135.496,E2 -14135.496} C_VEL
LIN {X 0,Y 339.402,Z 465.464,A -85,B 0,C 180,E1 -14137.138,E2 -14137.138} C_VEL
LIN {X 0,Y 339.69,Z 462.054,A -85,B 0,C 180,E1 -14138.329,E2 -14138.329} C_VEL
LIN {X 0,Y 340.2,Z 456.752,A -85,B 0,C 180,E1 -14139.814,E2 -14139.814} C_VEL
LIN {X 0,Y 340.741,Z 451.579,A -85,B 0,C 180,E1 -14141,E2 -14141} C_VEL
LIN {X 0,Y 341.454,Z 445.379,A -85,B 0,C 180,E1 -14142.181,E2 -14142.181} C_VEL
LIN {X 0,Y 342.151,Z 438.895,A -85,B 0,C 180,E1 -14143.211,E2 -14143.211} C_VEL
LIN {X 0,Y 343.014,Z 431.089,A -85,B 0,C 180,E1 -14144.235,E2 -14144.235} C_VEL
LIN {X 0,Y 343.314,Z 424.661,A -85,B 0,C 180,E1 -14144.953,E2 -14144.953} C_VEL
LIN {X 0,Y 343.022,Z 416.017,A -85,B 0,C 180,E1 -14145.783,E2 -14145.783} C_VEL
LIN {X 0,Y 342.071,Z 406.199,A -85,B 0,C 180,E1 -14146.564,E2 -14146.564} C_VEL
LIN {X 0,Y 340.367,Z 395.46,A -85,B 0,C 180,E1 -14147.253,E2 -14147.253} C_VEL
LIN {X 0,Y 339.693,Z 391.688,A -85,B 0,C 180,E1 -14147.453,E2 -14147.453} C_VEL
LIN {X 0,Y 340.259,Z 383.814,A -85,B 0,C 180,E1 -14151.647,E2 -14151.647} C_VEL
LIN {X 0,Y 340.931,Z 376.551,A -85,B 0,C 180,E1 -14155.653,E2 -14155.653} C_VEL
LIN {X 0,Y 341.602,Z 370.861,A -85,B 0,C 180,E1 -14158.914,E2 -14158.914} C_VEL
LIN {X 0,Y 342.438,Z 365.274,A -85,B 0,C 180,E1 -14162.251,E2 -14162.251} C_VEL
LIN {X 0,Y 342.633,Z 363.043,A -85,B 0,C 180,E1 -14163.631,E2 -14163.631} C_VEL
LIN {X 0,Y 342.241,Z 359.805,A -85,B 0,C 180,E1 -14165.822,E2 -14165.822} C_VEL
LIN {X 0,Y 341.419,Z 354.52,A -85,B 0,C 180,E1 -14169.654,E2 -14169.654} C_VEL
LIN {X 0,Y 340.726,Z 350.866,A -85,B 0,C 180,E1 -14172.662,E2 -14172.662} C_VEL
LIN {X 0,Y 340.683,Z 350.863,A -85,B 0,C 180,E1 -14177.096,E2 -14177.096} C_VEL
LIN {X 0,Y 340.707,Z 350.86,A -85,B 0,C 180,E1 -14180.248,E2 -14180.248} C_VEL
LIN {X 0,Y 340.717,Z 350.858,A -85,B 0,C 180,E1 -14183.56,E2 -14183.56} C_VEL
LIN {X 0,Y 340.7,Z 350.86,A -85,B 0,C 180,E1 -14186.153,E2 -14186.153} C_VEL
LIN {X 0,Y 340.749,Z 350.854,A -85,B 0,C 180,E1 -14190.329,E2 -14190.329} C_VEL
LIN {X 0,Y 340.811,Z 350.847,A -85,B 0,C 180,E1 -14193.02,E2 -14193.02} C_VEL
LIN {X 0,Y 340.764,Z 350.852,A -85,B 0,C 180,E1 -14195.638,E2 -14195.638} C_VEL
LIN {X 0,Y 340.761,Z 350.852,A -85,B 0,C 180,E1 -14199.474,E2 -14199.474} C_VEL
LIN {X 0,Y 340.866,Z 350.839,A -85,B 0,C 180,E1 -14201.984,E2 -14201.984} C_VEL
LIN {X 0,Y 340.877,Z 350.838,A -85,B 0,C 180,E1 -14205.704,E2 -14205.704} C_VEL
LIN {X 0,Y 340.855,Z 350.84,A -85,B 0,C 180,E1 -14209.305,E2 -14209.305} C_VEL
LIN {X 0,Y 341.023,Z 350.821,A -85,B 0,C 180,E1 -14212.896,E2 -14212.896} C_VEL
LIN {X 0,Y 341.17,Z 350.802,A -85,B 0,C 180,E1 -14217.638,E2 -14217.638} C_VEL
LIN {X 0,Y 341.282,Z 350.789,A -85,B 0,C 180,E1 -14219.999,E2 -14219.999} C_VEL
LIN {X 0,Y 341.173,Z 350.802,A -85,B 0,C 180,E1 -14222.36,E2 -14222.36} C_VEL
LIN {X 0,Y 341.051,Z 350.816,A -85,B 0,C 180,E1 -14227.101,E2 -14227.101} C_VEL
LIN {X 0,Y 340.852,Z 350.841,A -85,B 0,C 180,E1 -14230.693,E2 -14230.693} C_VEL
LIN {X 0,Y 340.867,Z 350.844,A -85,B 0,C 180,E1 -14234.323,E2 -14234.323} C_VEL
LIN {X 0,Y 340.593,Z 350.876,A -85,B 0,C 180,E1 -14238.029,E2 -14238.029} C_VEL
LIN {X 0,Y 340.378,Z 354.256,A -85,B 0,C 180,E1 -14241.816,E2 -14241.816} C_VEL
LIN {X 0,Y 340.092,Z 357.892,A -85,B 0,C 180,E1 -14245.718,E2 -14245.718} C_VEL
LIN {X 0,Y 339.935,Z 360.471,A -85,B 0,C 180,E1 -14248.391,E2 -14248.391} C_VEL
LIN {X 0,Y 339.687,Z 364.722,A -85,B 0,C 180,E1 -14252.673,E2 -14252.673} C_VEL
LIN {X 0,Y 342.598,Z 375.851,A -85,B 0,C 180,E1 -14253.455,E2 -14253.455} C_VEL
LIN {X 0,Y 344.253,Z 384.386,A -85,B 0,C 180,E1 -14254.18,E2 -14254.18} C_VEL
LIN {X 0,Y 345.02,Z 390.607,A -85,B 0,C 180,E1 -14254.773,E2 -14254.773} C_VEL
LIN {X 0,Y 344.149,Z 400.17,A -85,B 0,C 180,E1 -14255.786,E2 -14255.786} C_VEL
LIN {X 0,Y 343.367,Z 407.12,A -85,B 0,C 180,E1 -14256.684,E2 -14256.684} C_VEL
LIN {X 0,Y 342.723,Z 413.655,A -85,B 0,C 180,E1 -14257.707,E2 -14257.707} C_VEL
LIN {X 0,Y 341.993,Z 419.691,A -85,B 0,C 180,E1 -14258.837,E2 -14258.837} C_VEL
LIN {X 0,Y 341.365,Z 424.832,A -85,B 0,C 180,E1 -14259.991,E2 -14259.991} C_VEL
LIN {X 0,Y 340.765,Z 429.615,A -85,B 0,C 180,E1 -14261.296,E2 -14261.296} C_VEL
LIN {X 0,Y 340.129,Z 434.473,A -85,B 0,C 180,E1 -14262.988,E2 -14262.988} C_VEL
LIN {X 0,Y 339.787,Z 437.19,A -85,B 0,C 180,E1 -14264.219,E2 -14264.219} C_VEL
LIN {X 0,Y 339.539,Z 439.064,A -85,B 0,C 180,E1 -14265.269,E2 -14265.269} C_VEL
LIN {X 0,Y 339.226,Z 441.003,A -85,B 0,C 180,E1 -14266.866,E2 -14266.866} C_VEL
LIN {X 0,Y 339.037,Z 442.016,A -85,B 0,C 180,E1 -14268.444,E2 -14268.444} C_VEL
LIN {X 0,Y 338.986,Z 442.125,A -85,B 0,C 180,E1 -14270.092,E2 -14270.092} C_VEL
LIN {X 0,Y 339.03,Z 441.081,A -85,B 0,C 180,E1 -14271.971,E2 -14271.971} C_VEL
LIN {X 0,Y 339.281,Z 438.754,A -85,B 0,C 180,E1 -14273.885,E2 -14273.885} C_VEL
LIN {X 0,Y 339.583,Z 434.731,A -85,B 0,C 180,E1 -14275.874,E2 -14275.874} C_VEL
LIN {X 0,Y 340.02,Z 430.158,A -85,B 0,C 180,E1 -14277.491,E2 -14277.491} C_VEL
LIN {X 0,Y 340.473,Z 424.974,A -85,B 0,C 180,E1 -14278.931,E2 -14278.931} C_VEL
LIN {X 0,Y 340.913,Z 420.416,A -85,B 0,C 180,E1 -14279.975,E2 -14279.975} C_VEL
LIN {X 0,Y 341.478,Z 413.772,A -85,B 0,C 180,E1 -14281.242,E2 -14281.242} C_VEL
LIN {X 0,Y 342.057,Z 407.128,A -85,B 0,C 180,E1 -14282.288,E2 -14282.288} C_VEL
LIN {X 0,Y 342.705,Z 399.086,A -85,B 0,C 180,E1 -14283.332,E2 -14283.332} C_VEL
LIN {X 0,Y 343.405,Z 389.362,A -85,B 0,C 180,E1 -14284.343,E2 -14284.343} C_VEL
LIN {X 0,Y 343.374,Z 385.212,A -85,B 0,C 180,E1 -14284.695,E2 -14284.695} C_VEL
LIN {X 0,Y 342.043,Z 377.021,A -85,B 0,C 180,E1 -14285.354,E2 -14285.354} C_VEL
LIN {X 0,Y 340.355,Z 368.027,A -85,B 0,C 180,E1 -14285.931,E2 -14285.931} C_VEL
LIN {X 0,Y 339.442,Z 363.42,A -85,B 0,C 180,E1 -14286.186,E2 -14286.186} C_VEL
LIN {X 0,Y 339.528,Z 359.911,A -85,B 0,C 180,E1 -14289.396,E2 -14289.396} C_VEL
LIN {X 0,Y 339.744,Z 355.879,A -85,B 0,C 180,E1 -14293.164,E2 -14293.164} C_VEL
LIN {X 0,Y 339.984,Z 351.995,A -85,B 0,C 180,E1 -14296.855,E2 -14296.855} C_VEL
LIN {X 0,Y 340.053,Z 350.941,A -85,B 0,C 180,E1 -14298.071,E2 -14298.071} C_VEL
LIN {X 0,Y 340.804,Z 350.844,A -85,B 0,C 180,E1 -14301.815,E2 -14301.815} C_VEL
LIN {X 0,Y 341.001,Z 350.822,A -85,B 0,C 180,E1 -14304.084,E2 -14304.084} C_VEL
LIN {X 0,Y 341.16,Z 350.8,A -85,B 0,C 180,E1 -14307.637,E2 -14307.637} C_VEL
LIN {X 0,Y 341.286,Z 350.787,A -85,B 0,C 180,E1 -14309.998,E2 -14309.998} C_VEL
LIN {X 0,Y 341.161,Z 350.802,A -85,B 0,C 180,E1 -14312.36,E2 -14312.36} C_VEL
LIN {X 0,Y 341.068,Z 350.81,A -85,B 0,C 180,E1 -14317.1,E2 -14317.1} C_VEL
LIN {X 0,Y 340.864,Z 350.836,A -85,B 0,C 180,E1 -14320.692,E2 -14320.692} C_VEL
LIN {X 0,Y 340.851,Z 350.838,A -85,B 0,C 180,E1 -14324.324,E2 -14324.324} C_VEL
LIN {X 0,Y 340.824,Z 350.841,A -85,B 0,C 180,E1 -14328.465,E2 -14328.465} C_VEL
LIN {X 0,Y 340.741,Z 350.854,A -85,B 0,C 180,E1 -14331.856,E2 -14331.856} C_VEL
LIN {X 0,Y 340.759,Z 350.853,A -85,B 0,C 180,E1 -14335.663,E2 -14335.663} C_VEL
LIN {X 0,Y 340.728,Z 350.852,A -85,B 0,C 180,E1 -14338.319,E2 -14338.319} C_VEL
LIN {X 0,Y 340.69,Z 350.86,A -85,B 0,C 180,E1 -14341.043,E2 -14341.043} C_VEL
LIN {X 0,Y 340.705,Z 350.86,A -85,B 0,C 180,E1 -14345.278,E2 -14345.278} C_VEL
LIN {X 0,Y 340.711,Z 350.855,A -85,B 0,C 180,E1 -14348.389,E2 -14348.389} C_VEL
LIN {X 0,Y 340.737,Z 350.851,A -85,B 0,C 180,E1 -14352.055,E2 -14352.055} C_VEL
LIN {X 0,Y 340.767,Z 350.849,A -85,B 0,C 180,E1 -14355.477,E2 -14355.477} C_VEL
LIN {X 0,Y 340.713,Z 350.855,A -85,B 0,C 180,E1 -14359.096,E2 -14359.096} C_VEL
LIN {X 0,Y 340.727,Z 350.853,A -85,B 0,C 180,E1 -14361.774,E2 -14361.774} C_VEL
LIN {X 0,Y 340.684,Z 350.859,A -85,B 0,C 180,E1 -14364.217,E2 -14364.217} C_VEL
LIN {X 0,Y 340.018,Z 350.946,A -85,B 0,C 180,E1 -14365.205,E2 -14365.205} C_VEL
LIN {X 0,Y 337.125,Z 351.306,A -85,B 0,C 180,E1 -14366.81,E2 -14366.81} C_VEL
LIN {X 0,Y 334.703,Z 351.604,A -85,B 0,C 180,E1 -14368.11,E2 -14368.11} C_VEL
LIN {X 0,Y 333.716,Z 351.728,A -85,B 0,C 180,E1 -14369.116,E2 -14369.116} C_VEL
LIN {X 0,Y 333.664,Z 351.731,A -85,B 0,C 180,E1 -14369.457,E2 -14369.457} C_VEL
LIN {X 0,Y 333.731,Z 351.727,A -85,B 0,C 180,E1 -14372.402,E2 -14372.402} C_VEL
LIN {X 0,Y 333.747,Z 351.723,A -85,B 0,C 180,E1 -14375.094,E2 -14375.094} C_VEL
LIN {X 0,Y 333.71,Z 351.727,A -85,B 0,C 180,E1 -14379.023,E2 -14379.023} C_VEL
LIN {X 0,Y 333.782,Z 351.718,A -85,B 0,C 180,E1 -14381.59,E2 -14381.59} C_VEL
LIN {X 0,Y 333.795,Z 351.716,A -85,B 0,C 180,E1 -14385.577,E2 -14385.577} C_VEL
LIN {X 0,Y 333.825,Z 351.712,A -85,B 0,C 180,E1 -14389.079,E2 -14389.079} C_VEL
LIN {X 0,Y 334.014,Z 351.689,A -85,B 0,C 180,E1 -14392.749,E2 -14392.749} C_VEL
LIN {X 0,Y 333.801,Z 351.715,A -85,B 0,C 180,E1 -14395.17,E2 -14395.17} C_VEL
LIN {X 0,Y 334.096,Z 351.68,A -85,B 0,C 180,E1 -14397.59,E2 -14397.59} C_VEL
LIN {X 0,Y 334.236,Z 351.666,A -85,B 0,C 180,E1 -14400.001,E2 -14400.001} C_VEL
LIN {X 0,Y 334.098,Z 351.679,A -85,B 0,C 180,E1 -14402.412,E2 -14402.412} C_VEL
LIN {X 0,Y 334.015,Z 351.69,A -85,B 0,C 180,E1 -14407.254,E2 -14407.254} C_VEL
LIN {X 0,Y 333.828,Z 351.712,A -85,B 0,C 180,E1 -14410.923,E2 -14410.923} C_VEL
LIN {X 0,Y 333.799,Z 351.715,A -85,B 0,C 180,E1 -14414.636,E2 -14414.636} C_VEL
LIN {X 0,Y 333.787,Z 351.717,A -85,B 0,C 180,E1 -14418.656,E2 -14418.656} C_VEL
LIN {X 0,Y 333.684,Z 351.73,A -85,B 0,C 180,E1 -14422.28,E2 -14422.28} C_VEL
LIN {X 0,Y 333.728,Z 351.724,A -85,B 0,C 180,E1 -14426.248,E2 -14426.248} C_VEL
LIN {X 0,Y 333.704,Z 351.73,A -85,B 0,C 180,E1 -14428.974,E2 -14428.974} C_VEL
LIN {X 0,Y 333.637,Z 351.737,A -85,B 0,C 180,E1 -14432.589,E2 -14432.589} C_VEL
LIN {X 0,Y 333.67,Z 351.731,A -85,B 0,C 180,E1 -14436.141,E2 -14436.141} C_VEL
LIN {X 0,Y 333.641,Z 351.739,A -85,B 0,C 180,E1 -14439.194,E2 -14439.194} C_VEL
LIN {X 0,Y 333.628,Z 351.739,A -85,B 0,C 180,E1 -14442.502,E2 -14442.502} C_VEL
LIN {X 0,Y 333.616,Z 351.738,A -85,B 0,C 180,E1 -14445.961,E2 -14445.961} C_VEL
LIN {X 0,Y 333.748,Z 351.82,A -85,B 0,C 180,E1 -14449.885,E2 -14449.885} C_VEL
LIN {X 0,Y 334.554,Z 356.509,A -85,B 0,C 180,E1 -14452.966,E2 -14452.966} C_VEL
LIN {X 0,Y 335.208,Z 360.557,A -85,B 0,C 180,E1 -14455.525,E2 -14455.525} C_VEL
LIN {X 0,Y 335.166,Z 364.157,A -85,B 0,C 180,E1 -14457.686,E2 -14457.686} C_VEL
LIN {X 0,Y 334.37,Z 370.088,A -85,B 0,C 180,E1 -14461.092,E2 -14461.092} C_VEL
LIN {X 0,Y 333.588,Z 377.203,A -85,B 0,C 180,E1 -14465.082,E2 -14465.082} C_VEL
LIN {X 0,Y 332.988,Z 384.306,A -85,B 0,C 180,E1 -14468.975,E2 -14468.975} C_VEL
LIN {X 0,Y 332.504,Z 391.361,A -85,B 0,C 180,E1 -14472.79,E2 -14472.79} C_VEL
LIN {X 0,Y 332.471,Z 392.705,A -85,B 0,C 180,E1 -14473.5,E2 -14473.5} C_VEL
LIN {X 0,Y 333.827,Z 404.68,A -85,B 0,C 180,E1 -14474.118,E2 -14474.118} C_VEL
LIN {X 0,Y 334.802,Z 415.62,A -85,B 0,C 180,E1 -14474.932,E2 -14474.932} C_VEL
LIN {X 0,Y 335.268,Z 424.255,A -85,B 0,C 180,E1 -14475.743,E2 -14475.743} C_VEL
LIN {X 0,Y 334.985,Z 431.114,A -85,B 0,C 180,E1 -14476.504,E2 -14476.504} C_VEL
LIN {X 0,Y 334.27,Z 438.998,A -85,B 0,C 180,E1 -14477.557,E2 -14477.557} C_VEL
LIN {X 0,Y 333.624,Z 446.389,A -85,B 0,C 180,E1 -14478.765,E2 -14478.765} C_VEL
LIN {X 0,Y 332.939,Z 453.89,A -85,B 0,C 180,E1 -14480.279,E2 -14480.279} C_VEL
LIN {X 0,Y 332.444,Z 460.748,A -85,B 0,C 180,E1 -14482.103,E2 -14482.103} C_VEL
LIN {X 0,Y 332.102,Z 465.935,A -85,B 0,C 180,E1 -14483.928,E2 -14483.928} C_VEL
LIN {X 0,Y 332.082,Z 469.736,A -85,B 0,C 180,E1 -14485.754,E2 -14485.754} C_VEL
LIN {X 0,Y 332.018,Z 472.196,A -85,B 0,C 180,E1 -14487.575,E2 -14487.575} C_VEL
LIN {X 0,Y 332.076,Z 473.145,A -85,B 0,C 180,E1 -14488.789,E2 -14488.789} C_VEL
LIN {X 0,Y 332.132,Z 473.548,A -85,B 0,C 180,E1 -14490.002,E2 -14490.002} C_VEL
LIN {X 0,Y 332.062,Z 473.472,A -85,B 0,C 180,E1 -14491.214,E2 -14491.214} C_VEL
LIN {X 0,Y 331.991,Z 472.926,A -85,B 0,C 180,E1 -14492.428,E2 -14492.428} C_VEL
LIN {X 0,Y 332.046,Z 471.877,A -85,B 0,C 180,E1 -14493.642,E2 -14493.642} C_VEL
LIN {X 0,Y 332.053,Z 470.217,A -85,B 0,C 180,E1 -14494.858,E2 -14494.858} C_VEL
LIN {X 0,Y 332.218,Z 466.797,A -85,B 0,C 180,E1 -14496.683,E2 -14496.683} C_VEL
LIN {X 0,Y 332.647,Z 461.892,A -85,B 0,C 180,E1 -14498.506,E2 -14498.506} C_VEL
LIN {X 0,Y 333.162,Z 456.626,A -85,B 0,C 180,E1 -14500.024,E2 -14500.024} C_VEL
LIN {X 0,Y 333.943,Z 450.065,A -85,B 0,C 180,E1 -14501.534,E2 -14501.534} C_VEL
LIN {X 0,Y 334.892,Z 441.918,A -85,B 0,C 180,E1 -14503.04,E2 -14503.04} C_VEL
LIN {X 0,Y 336.02,Z 432.452,A -85,B 0,C 180,E1 -14504.383,E2 -14504.383} C_VEL
LIN {X 0,Y 336.443,Z 425.227,A -85,B 0,C 180,E1 -14505.235,E2 -14505.235} C_VEL
LIN {X 0,Y 336.198,Z 416.854,A -85,B 0,C 180,E1 -14506.081,E2 -14506.081} C_VEL
LIN {X 0,Y 335.387,Z 408.073,A -85,B 0,C 180,E1 -14506.826,E2 -14506.826} C_VEL
LIN {X 0,Y 333.994,Z 398.57,A -85,B 0,C 180,E1 -14507.487,E2 -14507.487} C_VEL
LIN {X 0,Y 332.671,Z 391.329,A -85,B 0,C 180,E1 -14507.923,E2 -14507.923} C_VEL
LIN {X 0,Y 333.211,Z 384.113,A -85,B 0,C 180,E1 -14511.868,E2 -14511.868} C_VEL
LIN {X 0,Y 334,Z 376.423,A -85,B 0,C 180,E1 -14516.225,E2 -14516.225} C_VEL
LIN {X 0,Y 334.903,Z 369.64,A -85,B 0,C 180,E1 -14520.243,E2 -14520.243} C_VEL
LIN {X 0,Y 335.559,Z 365.049,A -85,B 0,C 180,E1 -14523.094,E2 -14523.094} C_VEL
LIN {X 0,Y 335.409,Z 361.952,A -85,B 0,C 180,E1 -14525.195,E2 -14525.195} C_VEL
LIN {X 0,Y 334.563,Z 356.652,A -85,B 0,C 180,E1 -14529.066,E2 -14529.066} C_VEL
LIN {X 0,Y 333.799,Z 352.396,A -85,B 0,C 180,E1 -14532.53,E2 -14532.53} C_VEL
LIN {X 0,Y 333.658,Z 351.746,A -85,B 0,C 180,E1 -14533.224,E2 -14533.224} C_VEL
LIN {X 0,Y 333.649,Z 351.74,A -85,B 0,C 180,E1 -14537.619,E2 -14537.619} C_VEL
LIN {X 0,Y 333.66,Z 351.737,A -85,B 0,C 180,E1 -14541.202,E2 -14541.202} C_VEL
LIN {X 0,Y 333.684,Z 351.734,A -85,B 0,C 180,E1 -14543.861,E2 -14543.861} C_VEL
LIN {X 0,Y 333.651,Z 351.738,A -85,B 0,C 180,E1 -14547.413,E2 -14547.413} C_VEL
LIN {X 0,Y 333.698,Z 351.731,A -85,B 0,C 180,E1 -14551.026,E2 -14551.026} C_VEL
LIN {X 0,Y 333.743,Z 351.727,A -85,B 0,C 180,E1 -14553.753,E2 -14553.753} C_VEL
LIN {X 0,Y 333.728,Z 351.728,A -85,B 0,C 180,E1 -14557.914,E2 -14557.914} C_VEL
LIN {X 0,Y 333.802,Z 351.719,A -85,B 0,C 180,E1 -14561.589,E2 -14561.589} C_VEL
LIN {X 0,Y 333.816,Z 351.718,A -85,B 0,C 180,E1 -14565.576,E2 -14565.576} C_VEL
LIN {X 0,Y 333.825,Z 351.716,A -85,B 0,C 180,E1 -14569.077,E2 -14569.077} C_VEL
LIN {X 0,Y 333.975,Z 351.698,A -85,B 0,C 180,E1 -14572.745,E2 -14572.745} C_VEL
LIN {X 0,Y 333.802,Z 351.719,A -85,B 0,C 180,E1 -14575.168,E2 -14575.168} C_VEL
LIN {X 0,Y 334.107,Z 351.682,A -85,B 0,C 180,E1 -14577.588,E2 -14577.588} C_VEL
LIN {X 0,Y 334.234,Z 351.667,A -85,B 0,C 180,E1 -14579.999,E2 -14579.999} C_VEL
LIN {X 0,Y 334.11,Z 351.682,A -85,B 0,C 180,E1 -14582.41,E2 -14582.41} C_VEL
LIN {X 0,Y 333.987,Z 351.694,A -85,B 0,C 180,E1 -14586.606,E2 -14586.606} C_VEL
LIN {X 0,Y 333.825,Z 351.717,A -85,B 0,C 180,E1 -14589.695,E2 -14589.695} C_VEL
LIN {X 0,Y 333.797,Z 351.723,A -85,B 0,C 180,E1 -14593.39,E2 -14593.39} C_VEL
LIN {X 0,Y 333.702,Z 351.737,A -85,B 0,C 180,E1 -14595.888,E2 -14595.888} C_VEL
LIN {X 0,Y 333.595,Z 351.75,A -85,B 0,C 180,E1 -14597.153,E2 -14597.153} C_VEL
LIN {X 0,Y 333.533,Z 352.375,A -85,B 0,C 180,E1 -14598.517,E2 -14598.517} C_VEL
LIN {X 0,Y 333.296,Z 355.714,A -85,B 0,C 180,E1 -14602.305,E2 -14602.305} C_VEL
LIN {X 0,Y 333.002,Z 359.4,A -85,B 0,C 180,E1 -14606.307,E2 -14606.307} C_VEL
LIN {X 0,Y 332.762,Z 362.935,A -85,B 0,C 180,E1 -14610.009,E2 -14610.009} C_VEL
LIN {X 0,Y 332.653,Z 365.085,A -85,B 0,C 180,E1 -14612.208,E2 -14612.208} C_VEL
LIN {X 0,Y 335.527,Z 375.872,A -85,B 0,C 180,E1 -14612.995,E2 -14612.995} C_VEL
LIN {X 0,Y 337.431,Z 385.22,A -85,B 0,C 180,E1 -14613.821,E2 -14613.821} C_VEL
LIN {X 0,Y 338.217,Z 391.878,A -85,B 0,C 180,E1 -14614.487,E2 -14614.487} C_VEL
LIN {X 0,Y 337.422,Z 400.222,A -85,B 0,C 180,E1 -14615.389,E2 -14615.389} C_VEL
LIN {X 0,Y 336.582,Z 407.39,A -85,B 0,C 180,E1 -14616.332,E2 -14616.332} C_VEL
LIN {X 0,Y 335.783,Z 414.942,A -85,B 0,C 180,E1 -14617.558,E2 -14617.558} C_VEL
LIN {X 0,Y 335.078,Z 420.327,A -85,B 0,C 180,E1 -14618.605,E2 -14618.605} C_VEL
LIN {X 0,Y 334.377,Z 425.73,A -85,B 0,C 180,E1 -14619.868,E2 -14619.868} C_VEL
LIN {X 0,Y 333.753,Z 430.3,A -85,B 0,C 180,E1 -14621.164,E2 -14621.164} C_VEL
LIN {X 0,Y 333.248,Z 433.978,A -85,B 0,C 180,E1 -14622.441,E2 -14622.441} C_VEL
LIN {X 0,Y 332.746,Z 437.645,A -85,B 0,C 180,E1 -14624.099,E2 -14624.099} C_VEL
LIN {X 0,Y 332.349,Z 440.229,A -85,B 0,C 180,E1 -14625.745,E2 -14625.745} C_VEL
LIN {X 0,Y 331.998,Z 442.152,A -85,B 0,C 180,E1 -14627.806,E2 -14627.806} C_VEL
LIN {X 0,Y 331.9,Z 442.573,A -85,B 0,C 180,E1 -14629.665,E2 -14629.665} C_VEL
LIN {X 0,Y 331.93,Z 441.734,A -85,B 0,C 180,E1 -14631.571,E2 -14631.571} C_VEL
LIN {X 0,Y 332.147,Z 439.419,A -85,B 0,C 180,E1 -14633.667,E2 -14633.667} C_VEL
LIN {X 0,Y 332.463,Z 436.055,A -85,B 0,C 180,E1 -14635.527,E2 -14635.527} C_VEL
LIN {X 0,Y 332.866,Z 431.762,A -85,B 0,C 180,E1 -14637.19,E2 -14637.19} C_VEL
LIN {X 0,Y 333.368,Z 425.923,A -85,B 0,C 180,E1 -14638.901,E2 -14638.901} C_VEL
LIN {X 0,Y 333.837,Z 421.168,A -85,B 0,C 180,E1 -14640.036,E2 -14640.036} C_VEL
LIN {X 0,Y 334.434,Z 414.751,A -85,B 0,C 180,E1 -14641.303,E2 -14641.303} C_VEL
LIN {X 0,Y 335.083,Z 407.223,A -85,B 0,C 180,E1 -14642.519,E2 -14642.519} C_VEL
LIN {X 0,Y 335.786,Z 399.077,A -85,B 0,C 180,E1 -14643.59,E2 -14643.59} C_VEL
LIN {X 0,Y 336.547,Z 388.167,A -85,B 0,C 180,E1 -14644.718,E2 -14644.718} C_VEL
LIN {X 0,Y 335.249,Z 378.87,A -85,B 0,C 180,E1 -14645.51,E2 -14645.51} C_VEL
LIN {X 0,Y 333.321,Z 368.594,A -85,B 0,C 180,E1 -14646.2,E2 -14646.2} C_VEL
LIN {X 0,Y 332.353,Z 363.729,A -85,B 0,C 180,E1 -14646.474,E2 -14646.474} C_VEL
LIN {X 0,Y 332.487,Z 359.703,A -85,B 0,C 180,E1 -14650.231,E2 -14650.231} C_VEL
LIN {X 0,Y 332.67,Z 356.98,A -85,B 0,C 180,E1 -14652.795,E2 -14652.795} C_VEL
LIN {X 0,Y 332.916,Z 353.056,A -85,B 0,C 180,E1 -14656.571,E2 -14656.571} C_VEL
LIN {X 0,Y 332.979,Z 351.822,A -85,B 0,C 180,E1 -14657.814,E2 -14657.814} C_VEL
LIN {X 0,Y 333.744,Z 351.723,A -85,B 0,C 180,E1 -14661.768,E2 -14661.768} C_VEL
LIN {X 0,Y 333.969,Z 351.697,A -85,B 0,C 180,E1 -14663.959,E2 -14663.959} C_VEL
LIN {X 0,Y 334.097,Z 351.679,A -85,B 0,C 180,E1 -14667.587,E2 -14667.587} C_VEL
LIN {X 0,Y 334.237,Z 351.665,A -85,B 0,C 180,E1 -14669.998,E2 -14669.998} C_VEL
LIN {X 0,Y 334.098,Z 351.681,A -85,B 0,C 180,E1 -14672.41,E2 -14672.41} C_VEL
LIN {X 0,Y 334.014,Z 351.694,A -85,B 0,C 180,E1 -14676.037,E2 -14676.037} C_VEL
LIN {X 0,Y 333.973,Z 351.695,A -85,B 0,C 180,E1 -14678.5,E2 -14678.5} C_VEL
LIN {X 0,Y 333.784,Z 351.72,A -85,B 0,C 180,E1 -14682.153,E2 -14682.153} C_VEL
LIN {X 0,Y 333.765,Z 351.724,A -85,B 0,C 180,E1 -14685.885,E2 -14685.885} C_VEL
LIN {X 0,Y 333.783,Z 351.717,A -85,B 0,C 180,E1 -14688.654,E2 -14688.654} C_VEL
LIN {X 0,Y 333.679,Z 351.731,A -85,B 0,C 180,E1 -14692.277,E2 -14692.277} C_VEL
LIN {X 0,Y 333.722,Z 351.725,A -85,B 0,C 180,E1 -14696.245,E2 -14696.245} C_VEL
LIN {X 0,Y 333.698,Z 351.73,A -85,B 0,C 180,E1 -14698.971,E2 -14698.971} C_VEL
LIN {X 0,Y 333.629,Z 351.737,A -85,B 0,C 180,E1 -14702.586,E2 -14702.586} C_VEL
LIN {X 0,Y 333.664,Z 351.732,A -85,B 0,C 180,E1 -14706.138,E2 -14706.138} C_VEL
LIN {X 0,Y 333.673,Z 351.736,A -85,B 0,C 180,E1 -14709.186,E2 -14709.186} C_VEL
LIN {X 0,Y 333.688,Z 351.73,A -85,B 0,C 180,E1 -14712.513,E2 -14712.513} C_VEL
LIN {X 0,Y 333.714,Z 351.726,A -85,B 0,C 180,E1 -14715.977,E2 -14715.977} C_VEL
LIN {X 0,Y 333.687,Z 351.731,A -85,B 0,C 180,E1 -14719.304,E2 -14719.304} C_VEL
LIN {X 0,Y 333.653,Z 351.736,A -85,B 0,C 180,E1 -14723.167,E2 -14723.167} C_VEL
LIN {X 0,Y 333.622,Z 351.743,A -85,B 0,C 180,E1 -14726.792,E2 -14726.792} C_VEL
LIN {X 0,Y 333.664,Z 351.731,A -85,B 0,C 180,E1 -14729.457,E2 -14729.457} C_VEL
LIN {X 0,Y 333.08,Z 351.809,A -85,B 0,C 180,E1 -14730.465,E2 -14730.465} C_VEL
LIN {X 0,Y 330.275,Z 352.166,A -85,B 0,C 180,E1 -14732.105,E2 -14732.105} C_VEL
LIN {X 0,Y 327.836,Z 352.47,A -85,B 0,C 180,E1 -14733.433,E2 -14733.433} C_VEL
LIN {X 0,Y 326.766,Z 352.597,A -85,B 0,C 180,E1 -14734.461,E2 -14734.461} C_VEL
LIN {X 0,Y 326.669,Z 352.607,A -85,B 0,C 180,E1 -14734.81,E2 -14734.81} C_VEL
LIN {X 0,Y 326.662,Z 352.609,A -85,B 0,C 180,E1 -14738.548,E2 -14738.548} C_VEL
LIN {X 0,Y 326.731,Z 352.596,A -85,B 0,C 180,E1 -14741.178,E2 -14741.178} C_VEL
LIN {X 0,Y 326.75,Z 352.593,A -85,B 0,C 180,E1 -14745.434,E2 -14745.434} C_VEL
LIN {X 0,Y 326.761,Z 352.593,A -85,B 0,C 180,E1 -14748.84,E2 -14748.84} C_VEL
LIN {X 0,Y 326.967,Z 352.568,A -85,B 0,C 180,E1 -14752.591,E2 -14752.591} C_VEL
LIN {X 0,Y 326.768,Z 352.591,A -85,B 0,C 180,E1 -14755.066,E2 -14755.066} C_VEL
LIN {X 0,Y 327.037,Z 352.559,A -85,B 0,C 180,E1 -14757.538,E2 -14757.538} C_VEL
LIN {X 0,Y 327.187,Z 352.544,A -85,B 0,C 180,E1 -14760.001,E2 -14760.001} C_VEL
LIN {X 0,Y 327.039,Z 352.558,A -85,B 0,C 180,E1 -14762.464,E2 -14762.464} C_VEL
LIN {X 0,Y 326.986,Z 352.566,A -85,B 0,C 180,E1 -14766.17,E2 -14766.17} C_VEL
LIN {X 0,Y 326.905,Z 352.574,A -85,B 0,C 180,E1 -14768.656,E2 -14768.656} C_VEL
LIN {X 0,Y 326.729,Z 352.596,A -85,B 0,C 180,E1 -14772.423,E2 -14772.423} C_VEL
LIN {X 0,Y 326.745,Z 352.594,A -85,B 0,C 180,E1 -14774.959,E2 -14774.959} C_VEL
LIN {X 0,Y 326.724,Z 352.597,A -85,B 0,C 180,E1 -14778.84,E2 -14778.84} C_VEL
LIN {X 0,Y 326.613,Z 352.611,A -85,B 0,C 180,E1 -14782.789,E2 -14782.789} C_VEL
LIN {X 0,Y 326.682,Z 352.606,A -85,B 0,C 180,E1 -14785.485,E2 -14785.485} C_VEL
LIN {X 0,Y 326.654,Z 352.607,A -85,B 0,C 180,E1 -14789.661,E2 -14789.661} C_VEL
LIN {X 0,Y 326.6,Z 352.612,A -85,B 0,C 180,E1 -14794.021,E2 -14794.021} C_VEL
LIN {X 0,Y 326.622,Z 352.613,A -85,B 0,C 180,E1 -14797.24,E2 -14797.24} C_VEL
LIN {X 0,Y 326.572,Z 352.619,A -85,B 0,C 180,E1 -14801.133,E2 -14801.133} C_VEL
LIN {X 0,Y 326.552,Z 352.622,A -85,B 0,C 180,E1 -14804.75,E2 -14804.75} C_VEL
LIN {X 0,Y 326.585,Z 352.614,A -85,B 0,C 180,E1 -14808.158,E2 -14808.158} C_VEL
LIN {X 0,Y 326.701,Z 352.725,A -85,B 0,C 180,E1 -14809.694,E2 -14809.694} C_VEL
LIN {X 0,Y 327.574,Z 357.771,A -85,B 0,C 180,E1 -14813.08,E2 -14813.08} C_VEL
LIN {X 0,Y 328.28,Z 362.6,A -85,B 0,C 180,E1 -14816.18,E2 -14816.18} C_VEL
LIN {X 0,Y 327.931,Z 366.171,A -85,B 0,C 180,E1 -14818.329,E2 -14818.329} C_VEL
LIN {X 0,Y 327.029,Z 373.28,A -85,B 0,C 180,E1 -14822.483,E2 -14822.483} C_VEL
LIN {X 0,Y 326.252,Z 380.36,A -85,B 0,C 180,E1 -14826.516,E2 -14826.516} C_VEL
LIN {X 0,Y 325.754,Z 386.235,A -85,B 0,C 180,E1 -14829.808,E2 -14829.808} C_VEL
LIN {X 0,Y 325.402,Z 392.347,A -85,B 0,C 180,E1 -14833.171,E2 -14833.171} C_VEL
LIN {X 0,Y 326.913,Z 405.798,A -85,B 0,C 180,E1 -14833.936,E2 -14833.936} C_VEL
LIN {X 0,Y 327.697,Z 414.58,A -85,B 0,C 180,E1 -14834.604,E2 -14834.604} C_VEL
LIN {X 0,Y 328.218,Z 423.294,A -85,B 0,C 180,E1 -14835.43,E2 -14835.43} C_VEL
LIN {X 0,Y 328.063,Z 430.28,A -85,B 0,C 180,E1 -14836.214,E2 -14836.214} C_VEL
LIN {X 0,Y 327.233,Z 438.238,A -85,B 0,C 180,E1 -14837.285,E2 -14837.285} C_VEL
LIN {X 0,Y 326.772,Z 443.995,A -85,B 0,C 180,E1 -14838.212,E2 -14838.212} C_VEL
LIN {X 0,Y 326.16,Z 450.418,A -85,B 0,C 180,E1 -14839.448,E2 -14839.448} C_VEL
LIN {X 0,Y 325.725,Z 455.763,A -85,B 0,C 180,E1 -14840.689,E2 -14840.689} C_VEL
LIN {X 0,Y 325.38,Z 460.218,A -85,B 0,C 180,E1 -14841.931,E2 -14841.931} C_VEL
LIN {X 0,Y 325.045,Z 465.447,A -85,B 0,C 180,E1 -14843.795,E2 -14843.795} C_VEL
LIN {X 0,Y 324.994,Z 469.285,A -85,B 0,C 180,E1 -14845.661,E2 -14845.661} C_VEL
LIN {X 0,Y 324.932,Z 471.803,A -85,B 0,C 180,E1 -14847.522,E2 -14847.522} C_VEL
LIN {X 0,Y 324.981,Z 472.761,A -85,B 0,C 180,E1 -14848.762,E2 -14848.762} C_VEL
LIN {X 0,Y 325.04,Z 473.196,A -85,B 0,C 180,E1 -14850.002,E2 -14850.002} C_VEL
LIN {X 0,Y 324.964,Z 473.151,A -85,B 0,C 180,E1 -14851.241,E2 -14851.241} C_VEL
LIN {X 0,Y 324.907,Z 472.635,A -85,B 0,C 180,E1 -14852.481,E2 -14852.481} C_VEL
LIN {X 0,Y 324.972,Z 471.597,A -85,B 0,C 180,E1 -14853.721,E2 -14853.721} C_VEL
LIN {X 0,Y 324.977,Z 468.495,A -85,B 0,C 180,E1 -14855.839,E2 -14855.839} C_VEL
LIN {X 0,Y 325.296,Z 465.067,A -85,B 0,C 180,E1 -14857.45,E2 -14857.45} C_VEL
LIN {X 0,Y 325.809,Z 459.789,A -85,B 0,C 180,E1 -14859.312,E2 -14859.312} C_VEL
LIN {X 0,Y 326.611,Z 452.882,A -85,B 0,C 180,E1 -14861.168,E2 -14861.168} C_VEL
LIN {X 0,Y 327.581,Z 445.385,A -85,B 0,C 180,E1 -14862.705,E2 -14862.705} C_VEL
LIN {X 0,Y 328.472,Z 438.036,A -85,B 0,C 180,E1 -14863.93,E2 -14863.93} C_VEL
LIN {X 0,Y 329.39,Z 430.361,A -85,B 0,C 180,E1 -14864.976,E2 -14864.976} C_VEL
LIN {X 0,Y 329.56,Z 423.46,A -85,B 0,C 180,E1 -14865.788,E2 -14865.788} C_VEL
LIN {X 0,Y 329.183,Z 415.545,A -85,B 0,C 180,E1 -14866.593,E2 -14866.593} C_VEL
LIN {X 0,Y 328.323,Z 406.525,A -85,B 0,C 180,E1 -14867.36,E2 -14867.36} C_VEL
LIN {X 0,Y 326.619,Z 396.046,A -85,B 0,C 180,E1 -14868.093,E2 -14868.093} C_VEL
LIN {X 0,Y 325.636,Z 390.97,A -85,B 0,C 180,E1 -14868.403,E2 -14868.403} C_VEL
LIN {X 0,Y 326.176,Z 384.405,A -85,B 0,C 180,E1 -14872.102,E2 -14872.102} C_VEL
LIN {X 0,Y 326.93,Z 377.428,A -85,B 0,C 180,E1 -14876.149,E2 -14876.149} C_VEL
LIN {X 0,Y 327.861,Z 370.703,A -85,B 0,C 180,E1 -14880.25,E2 -14880.25} C_VEL
LIN {X 0,Y 328.409,Z 367.362,A -85,B 0,C 180,E1 -14882.346,E2 -14882.346} C_VEL
LIN {X 0,Y 328.522,Z 364.111,A -85,B 0,C 180,E1 -14884.537,E2 -14884.537} C_VEL
LIN {X 0,Y 327.7,Z 358.784,A -85,B 0,C 180,E1 -14888.46,E2 -14888.46} C_VEL
LIN {X 0,Y 327.004,Z 354.735,A -85,B 0,C 180,E1 -14891.78,E2 -14891.78} C_VEL
LIN {X 0,Y 326.594,Z 352.625,A -85,B 0,C 180,E1 -14893.735,E2 -14893.735} C_VEL
LIN {X 0,Y 326.584,Z 352.62,A -85,B 0,C 180,E1 -14897.028,E2 -14897.028} C_VEL
LIN {X 0,Y 326.619,Z 352.614,A -85,B 0,C 180,E1 -14900.773,E2 -14900.773} C_VEL
LIN {X 0,Y 326.62,Z 352.614,A -85,B 0,C 180,E1 -14904.48,E2 -14904.48} C_VEL
LIN {X 0,Y 326.616,Z 352.614,A -85,B 0,C 180,E1 -14907.455,E2 -14907.455} C_VEL
LIN {X 0,Y 326.656,Z 352.609,A -85,B 0,C 180,E1 -14910.339,E2 -14910.339} C_VEL
LIN {X 0,Y 326.698,Z 352.604,A -85,B 0,C 180,E1 -14914.516,E2 -14914.516} C_VEL
LIN {X 0,Y 326.657,Z 352.608,A -85,B 0,C 180,E1 -14918.545,E2 -14918.545} C_VEL
LIN {X 0,Y 326.753,Z 352.597,A -85,B 0,C 180,E1 -14921.177,E2 -14921.177} C_VEL
LIN {X 0,Y 326.771,Z 352.595,A -85,B 0,C 180,E1 -14925.432,E2 -14925.432} C_VEL
LIN {X 0,Y 326.765,Z 352.595,A -85,B 0,C 180,E1 -14928.838,E2 -14928.838} C_VEL
LIN {X 0,Y 326.93,Z 352.575,A -85,B 0,C 180,E1 -14932.588,E2 -14932.588} C_VEL
LIN {X 0,Y 326.769,Z 352.595,A -85,B 0,C 180,E1 -14935.064,E2 -14935.064} C_VEL
LIN {X 0,Y 327.048,Z 352.561,A -85,B 0,C 180,E1 -14937.536,E2 -14937.536} C_VEL
LIN {X 0,Y 327.186,Z 352.545,A -85,B 0,C 180,E1 -14939.999,E2 -14939.999} C_VEL
LIN {X 0,Y 327.051,Z 352.561,A -85,B 0,C 180,E1 -14942.462,E2 -14942.462} C_VEL
LIN {X 0,Y 326.956,Z 352.57,A -85,B 0,C 180,E1 -14946.595,E2 -14946.595} C_VEL
LIN {X 0,Y 326.788,Z 352.593,A -85,B 0,C 180,E1 -14949.906,E2 -14949.906} C_VEL
LIN {X 0,Y 326.76,Z 352.6,A -85,B 0,C 180,E1 -14953.684,E2 -14953.684} C_VEL
LIN {X 0,Y 326.623,Z 352.62,A -85,B 0,C 180,E1 -14956.242,E2 -14956.242} C_VEL
LIN {X 0,Y 326.513,Z 352.667,A -85,B 0,C 180,E1 -14957.537,E2 -14957.537} C_VEL
LIN {X 0,Y 326.401,Z 354.86,A -85,B 0,C 180,E1 -14960.15,E2 -14960.15} C_VEL
LIN {X 0,Y 326.211,Z 357.185,A -85,B 0,C 180,E1 -14962.816,E2 -14962.816} C_VEL
LIN {X 0,Y 326.015,Z 359.623,A -85,B 0,C 180,E1 -14965.539,E2 -14965.539} C_VEL
LIN {X 0,Y 325.818,Z 362.223,A -85,B 0,C 180,E1 -14968.328,E2 -14968.328} C_VEL
LIN {X 0,Y 325.659,Z 365.628,A -85,B 0,C 180,E1 -14971.736,E2 -14971.736} C_VEL
LIN {X 0,Y 328.683,Z 376.766,A -85,B 0,C 180,E1 -14972.59,E2 -14972.59} C_VEL
LIN {X 0,Y 330.586,Z 386.032,A -85,B 0,C 180,E1 -14973.443,E2 -14973.443} C_VEL
LIN {X 0,Y 331.468,Z 391.592,A -85,B 0,C 180,E1 -14974.02,E2 -14974.02} C_VEL
LIN {X 0,Y 330.695,Z 400.575,A -85,B 0,C 180,E1 -14975.014,E2 -14975.014} C_VEL
LIN {X 0,Y 329.752,Z 408.221,A -85,B 0,C 180,E1 -14976.048,E2 -14976.048} C_VEL
LIN {X 0,Y 328.962,Z 415.098,A -85,B 0,C 180,E1 -14977.188,E2 -14977.188} C_VEL
LIN {X 0,Y 327.981,Z 422.305,A -85,B 0,C 180,E1 -14978.652,E2 -14978.652} C_VEL
LIN {X 0,Y 327.199,Z 428.084,A -85,B 0,C 180,E1 -14980.117,E2 -14980.117} C_VEL
LIN {X 0,Y 326.366,Z 433.524,A -85,B 0,C 180,E1 -14981.877,E2 -14981.877} C_VEL
LIN {X 0,Y 325.802,Z 437.526,A -85,B 0,C 180,E1 -14983.65,E2 -14983.65} C_VEL
LIN {X 0,Y 325.35,Z 440.412,A -85,B 0,C 180,E1 -14985.464,E2 -14985.464} C_VEL
LIN {X 0,Y 325.18,Z 441.379,A -85,B 0,C 180,E1 -14986.241,E2 -14986.241} C_VEL
LIN {X 0,Y 324.899,Z 442.598,A -85,B 0,C 180,E1 -14987.887,E2 -14987.887} C_VEL
LIN {X 0,Y 324.809,Z 442.926,A -85,B 0,C 180,E1 -14989.523,E2 -14989.523} C_VEL
LIN {X 0,Y 324.843,Z 442.383,A -85,B 0,C 180,E1 -14991.154,E2 -14991.154} C_VEL
LIN {X 0,Y 324.965,Z 440.477,A -85,B 0,C 180,E1 -14993.146,E2 -14993.146} C_VEL
LIN {X 0,Y 325.173,Z 438.841,A -85,B 0,C 180,E1 -14994.298,E2 -14994.298} C_VEL
LIN {X 0,Y 325.412,Z 435.812,A -85,B 0,C 180,E1 -14995.837,E2 -14995.837} C_VEL
LIN {X 0,Y 325.927,Z 430.655,A -85,B 0,C 180,E1 -14997.744,E2 -14997.744} C_VEL
LIN {X 0,Y 326.387,Z 425.617,A -85,B 0,C 180,E1 -14999.196,E2 -14999.196} C_VEL
LIN {X 0,Y 326.887,Z 420.697,A -85,B 0,C 180,E1 -15000.362,E2 -15000.362} C_VEL
LIN {X 0,Y 327.485,Z 414.297,A -85,B 0,C 180,E1 -15001.624,E2 -15001.624} C_VEL
LIN {X 0,Y 328.126,Z 407.373,A -85,B 0,C 180,E1 -15002.752,E2 -15002.752} C_VEL
LIN {X 0,Y 328.921,Z 398.358,A -85,B 0,C 180,E1 -15003.949,E2 -15003.949} C_VEL
LIN {X 0,Y 329.599,Z 389.019,A -85,B 0,C 180,E1 -15004.924,E2 -15004.924} C_VEL
LIN {X 0,Y 328.468,Z 380.659,A -85,B 0,C 180,E1 -15005.676,E2 -15005.676} C_VEL
LIN {X 0,Y 326.429,Z 369.812,A -85,B 0,C 180,E1 -15006.442,E2 -15006.442} C_VEL
LIN {X 0,Y 325.288,Z 364.048,A -85,B 0,C 180,E1 -15006.776,E2 -15006.776} C_VEL
LIN {X 0,Y 325.38,Z 360.853,A -85,B 0,C 180,E1 -15009.781,E2 -15009.781} C_VEL
LIN {X 0,Y 325.585,Z 358.107,A -85,B 0,C 180,E1 -15012.409,E2 -15012.409} C_VEL
LIN {X 0,Y 325.848,Z 354.132,A -85,B 0,C 180,E1 -15016.274,E2 -15016.274} C_VEL
LIN {X 0,Y 325.917,Z 352.853,A -85,B 0,C 180,E1 -15017.546,E2 -15017.546} C_VEL
LIN {X 0,Y 326.681,Z 352.603,A -85,B 0,C 180,E1 -15021.722,E2 -15021.722} C_VEL
LIN {X 0,Y 326.916,Z 352.574,A -85,B 0,C 180,E1 -15023.828,E2 -15023.828} C_VEL
LIN {X 0,Y 327.038,Z 352.558,A -85,B 0,C 180,E1 -15027.535,E2 -15027.535} C_VEL
LIN {X 0,Y 327.189,Z 352.543,A -85,B 0,C 180,E1 -15029.998,E2 -15029.998} C_VEL
LIN {X 0,Y 327.039,Z 352.559,A -85,B 0,C 180,E1 -15032.462,E2 -15032.462} C_VEL
LIN {X 0,Y 326.989,Z 352.567,A -85,B 0,C 180,E1 -15036.168,E2 -15036.168} C_VEL
LIN {X 0,Y 326.904,Z 352.574,A -85,B 0,C 180,E1 -15038.654,E2 -15038.654} C_VEL
LIN {X 0,Y 326.727,Z 352.597,A -85,B 0,C 180,E1 -15042.42,E2 -15042.42} C_VEL
LIN {X 0,Y 326.742,Z 352.594,A -85,B 0,C 180,E1 -15044.956,E2 -15044.956} C_VEL
LIN {X 0,Y 326.72,Z 352.597,A -85,B 0,C 180,E1 -15048.837,E2 -15048.837} C_VEL
LIN {X 0,Y 326.608,Z 352.611,A -85,B 0,C 180,E1 -15052.786,E2 -15052.786} C_VEL
LIN {X 0,Y 326.677,Z 352.608,A -85,B 0,C 180,E1 -15055.483,E2 -15055.483} C_VEL
LIN {X 0,Y 326.647,Z 352.609,A -85,B 0,C 180,E1 -15059.658,E2 -15059.658} C_VEL
LIN {X 0,Y 326.593,Z 352.613,A -85,B 0,C 180,E1 -15064.019,E2 -15064.019} C_VEL
LIN {X 0,Y 326.619,Z 352.615,A -85,B 0,C 180,E1 -15067.239,E2 -15067.239} C_VEL
LIN {X 0,Y 326.622,Z 352.609,A -85,B 0,C 180,E1 -15070.202,E2 -15070.202} C_VEL
LIN {X 0,Y 326.643,Z 352.608,A -85,B 0,C 180,E1 -15073.509,E2 -15073.509} C_VEL
LIN {X 0,Y 326.635,Z 352.613,A -85,B 0,C 180,E1 -15077.014,E2 -15077.014} C_VEL
LIN {X 0,Y 326.631,Z 352.612,A -85,B 0,C 180,E1 -15080.765,E2 -15080.765} C_VEL
LIN {X 0,Y 326.599,Z 352.615,A -85,B 0,C 180,E1 -15084.481,E2 -15084.481} C_VEL
LIN {X 0,Y 326.594,Z 352.613,A -85,B 0,C 180,E1 -15087.456,E2 -15087.456} C_VEL
LIN {X 0,Y 326.647,Z 352.609,A -85,B 0,C 180,E1 -15090.341,E2 -15090.341} C_VEL
LIN {X 0,Y 326.68,Z 352.607,A -85,B 0,C 180,E1 -15094.517,E2 -15094.517} C_VEL
LIN {X 0,Y 326.669,Z 352.607,A -85,B 0,C 180,E1 -15094.81,E2 -15094.81} C_VEL
LIN {X 0,Y 325.968,Z 352.692,A -85,B 0,C 180,E1 -15095.839,E2 -15095.839} C_VEL
LIN {X 0,Y 323.089,Z 353.049,A -85,B 0,C 180,E1 -15097.513,E2 -15097.513} C_VEL
LIN {X 0,Y 320.693,Z 353.35,A -85,B 0,C 180,E1 -15098.87,E2 -15098.87} C_VEL
LIN {X 0,Y 319.702,Z 353.472,A -85,B 0,C 180,E1 -15099.92,E2 -15099.92} C_VEL
LIN {X 0,Y 319.64,Z 353.478,A -85,B 0,C 180,E1 -15100.276,E2 -15100.276} C_VEL
LIN {X 0,Y 319.662,Z 353.476,A -85,B 0,C 180,E1 -15103.394,E2 -15103.394} C_VEL
LIN {X 0,Y 319.72,Z 353.472,A -85,B 0,C 180,E1 -15106.009,E2 -15106.009} C_VEL
LIN {X 0,Y 319.748,Z 353.468,A -85,B 0,C 180,E1 -15109.874,E2 -15109.874} C_VEL
LIN {X 0,Y 319.921,Z 353.447,A -85,B 0,C 180,E1 -15112.427,E2 -15112.427} C_VEL
LIN {X 0,Y 319.737,Z 353.467,A -85,B 0,C 180,E1 -15114.957,E2 -15114.957} C_VEL
LIN {X 0,Y 319.981,Z 353.437,A -85,B 0,C 180,E1 -15117.484,E2 -15117.484} C_VEL
LIN {X 0,Y 320.139,Z 353.422,A -85,B 0,C 180,E1 -15120.001,E2 -15120.001} C_VEL
LIN {X 0,Y 319.983,Z 353.437,A -85,B 0,C 180,E1 -15122.519,E2 -15122.519} C_VEL
LIN {X 0,Y 319.942,Z 353.443,A -85,B 0,C 180,E1 -15126.307,E2 -15126.307} C_VEL
LIN {X 0,Y 319.833,Z 353.455,A -85,B 0,C 180,E1 -15128.849,E2 -15128.849} C_VEL
LIN {X 0,Y 319.675,Z 353.474,A -85,B 0,C 180,E1 -15132.701,E2 -15132.701} C_VEL
LIN {X 0,Y 319.69,Z 353.475,A -85,B 0,C 180,E1 -15135.297,E2 -15135.297} C_VEL
LIN {X 0,Y 319.665,Z 353.479,A -85,B 0,C 180,E1 -15139.257,E2 -15139.257} C_VEL
LIN {X 0,Y 319.562,Z 353.493,A -85,B 0,C 180,E1 -15143.321,E2 -15143.321} C_VEL
LIN {X 0,Y 319.627,Z 353.481,A -85,B 0,C 180,E1 -15146.09,E2 -15146.09} C_VEL
LIN {X 0,Y 319.583,Z 353.488,A -85,B 0,C 180,E1 -15148.935,E2 -15148.935} C_VEL
LIN {X 0,Y 319.526,Z 353.494,A -85,B 0,C 180,E1 -15151.864,E2 -15151.864} C_VEL
LIN {X 0,Y 319.574,Z 353.489,A -85,B 0,C 180,E1 -15155.545,E2 -15155.545} C_VEL
LIN {X 0,Y 319.553,Z 353.49,A -85,B 0,C 180,E1 -15159.671,E2 -15159.671} C_VEL
LIN {X 0,Y 319.552,Z 353.491,A -85,B 0,C 180,E1 -15163.469,E2 -15163.469} C_VEL
LIN {X 0,Y 319.556,Z 353.493,A -85,B 0,C 180,E1 -15167.02,E2 -15167.02} C_VEL
LIN {X 0,Y 319.634,Z 353.545,A -85,B 0,C 180,E1 -15169.447,E2 -15169.447} C_VEL
LIN {X 0,Y 320.536,Z 358.636,A -85,B 0,C 180,E1 -15172.956,E2 -15172.956} C_VEL
LIN {X 0,Y 321.234,Z 363.642,A -85,B 0,C 180,E1 -15176.241,E2 -15176.241} C_VEL
LIN {X 0,Y 320.795,Z 367.647,A -85,B 0,C 180,E1 -15178.696,E2 -15178.696} C_VEL
LIN {X 0,Y 319.935,Z 374.064,A -85,B 0,C 180,E1 -15182.531,E2 -15182.531} C_VEL
LIN {X 0,Y 319.247,Z 379.969,A -85,B 0,C 180,E1 -15185.969,E2 -15185.969} C_VEL
LIN {X 0,Y 318.742,Z 385.822,A -85,B 0,C 180,E1 -15189.344,E2 -15189.344} C_VEL
LIN {X 0,Y 318.315,Z 392.039,A -85,B 0,C 180,E1 -15192.868,E2 -15192.868} C_VEL
LIN {X 0,Y 319.863,Z 405.596,A -85,B 0,C 180,E1 -15193.651,E2 -15193.651} C_VEL
LIN {X 0,Y 320.588,Z 413.543,A -85,B 0,C 180,E1 -15194.262,E2 -15194.262} C_VEL
LIN {X 0,Y 321.142,Z 422.326,A -85,B 0,C 180,E1 -15195.101,E2 -15195.101} C_VEL
LIN {X 0,Y 321.141,Z 429.444,A -85,B 0,C 180,E1 -15195.911,E2 -15195.911} C_VEL
LIN {X 0,Y 320.297,Z 437.487,A -85,B 0,C 180,E1 -15197.004,E2 -15197.004} C_VEL
LIN {X 0,Y 319.773,Z 443.309,A -85,B 0,C 180,E1 -15197.95,E2 -15197.95} C_VEL
LIN {X 0,Y 319.141,Z 449.791,A -85,B 0,C 180,E1 -15199.213,E2 -15199.213} C_VEL
LIN {X 0,Y 318.698,Z 455.189,A -85,B 0,C 180,E1 -15200.482,E2 -15200.482} C_VEL
LIN {X 0,Y 318.316,Z 459.688,A -85,B 0,C 180,E1 -15201.751,E2 -15201.751} C_VEL
LIN {X 0,Y 318.081,Z 463.433,A -85,B 0,C 180,E1 -15203.022,E2 -15203.022} C_VEL
LIN {X 0,Y 317.879,Z 467.676,A -85,B 0,C 180,E1 -15204.928,E2 -15204.928} C_VEL
LIN {X 0,Y 317.92,Z 469.824,A -85,B 0,C 180,E1 -15206.199,E2 -15206.199} C_VEL
LIN {X 0,Y 317.85,Z 471.406,A -85,B 0,C 180,E1 -15207.467,E2 -15207.467} C_VEL
LIN {X 0,Y 317.886,Z 472.377,A -85,B 0,C 180,E1 -15208.735,E2 -15208.735} C_VEL
LIN {X 0,Y 317.948,Z 472.843,A -85,B 0,C 180,E1 -15210.002,E2 -15210.002} C_VEL
LIN {X 0,Y 317.868,Z 472.829,A -85,B 0,C 180,E1 -15211.269,E2 -15211.269} C_VEL
LIN {X 0,Y 317.826,Z 472.347,A -85,B 0,C 180,E1 -15212.536,E2 -15212.536} C_VEL
LIN {X 0,Y 317.876,Z 471.316,A -85,B 0,C 180,E1 -15213.805,E2 -15213.805} C_VEL
LIN {X 0,Y 317.873,Z 468.656,A -85,B 0,C 180,E1 -15215.769,E2 -15215.769} C_VEL
LIN {X 0,Y 318.235,Z 464.901,A -85,B 0,C 180,E1 -15217.616,E2 -15217.616} C_VEL
LIN {X 0,Y 318.77,Z 459.666,A -85,B 0,C 180,E1 -15219.519,E2 -15219.519} C_VEL
LIN {X 0,Y 319.477,Z 454.072,A -85,B 0,C 180,E1 -15221.099,E2 -15221.099} C_VEL
LIN {X 0,Y 320.405,Z 447.108,A -85,B 0,C 180,E1 -15222.672,E2 -15222.672} C_VEL
LIN {X 0,Y 321.586,Z 438.152,A -85,B 0,C 180,E1 -15224.234,E2 -15224.234} C_VEL
LIN {X 0,Y 322.525,Z 430.61,A -85,B 0,C 180,E1 -15225.297,E2 -15225.297} C_VEL
LIN {X 0,Y 322.661,Z 423.06,A -85,B 0,C 180,E1 -15226.215,E2 -15226.215} C_VEL
LIN {X 0,Y 322.353,Z 416.07,A -85,B 0,C 180,E1 -15226.955,E2 -15226.955} C_VEL
LIN {X 0,Y 321.536,Z 407.379,A -85,B 0,C 180,E1 -15227.738,E2 -15227.738} C_VEL
LIN {X 0,Y 320.077,Z 397.972,A -85,B 0,C 180,E1 -15228.445,E2 -15228.445} C_VEL
LIN {X 0,Y 318.622,Z 390.611,A -85,B 0,C 180,E1 -15228.937,E2 -15228.937} C_VEL
LIN {X 0,Y 319.131,Z 384.706,A -85,B 0,C 180,E1 -15232.339,E2 -15232.339} C_VEL
LIN {X 0,Y 319.868,Z 378.453,A -85,B 0,C 180,E1 -15236.069,E2 -15236.069} C_VEL
LIN {X 0,Y 320.84,Z 371.747,A -85,B 0,C 180,E1 -15240.254,E2 -15240.254} C_VEL
LIN {X 0,Y 321.52,Z 367.351,A -85,B 0,C 180,E1 -15243.126,E2 -15243.126} C_VEL
LIN {X 0,Y 321.503,Z 365.164,A -85,B 0,C 180,E1 -15244.637,E2 -15244.637} C_VEL
LIN {X 0,Y 320.831,Z 360.769,A -85,B 0,C 180,E1 -15247.944,E2 -15247.944} C_VEL
LIN {X 0,Y 320.192,Z 356.856,A -85,B 0,C 180,E1 -15251.186,E2 -15251.186} C_VEL
LIN {X 0,Y 319.519,Z 353.505,A -85,B 0,C 180,E1 -15254.225,E2 -15254.225} C_VEL
LIN {X 0,Y 319.562,Z 353.494,A -85,B 0,C 180,E1 -15257.017,E2 -15257.017} C_VEL
LIN {X 0,Y 319.555,Z 353.495,A -85,B 0,C 180,E1 -15260.371,E2 -15260.371} C_VEL
LIN {X 0,Y 319.566,Z 353.492,A -85,B 0,C 180,E1 -15263.572,E2 -15263.572} C_VEL
LIN {X 0,Y 319.585,Z 353.49,A -85,B 0,C 180,E1 -15266.686,E2 -15266.686} C_VEL
LIN {X 0,Y 319.593,Z 353.489,A -85,B 0,C 180,E1 -15269.616,E2 -15269.616} C_VEL
LIN {X 0,Y 319.614,Z 353.486,A -85,B 0,C 180,E1 -15272.498,E2 -15272.498} C_VEL
LIN {X 0,Y 319.613,Z 353.486,A -85,B 0,C 180,E1 -15275.304,E2 -15275.304} C_VEL
LIN {X 0,Y 319.606,Z 353.486,A -85,B 0,C 180,E1 -15278.047,E2 -15278.047} C_VEL
LIN {X 0,Y 319.697,Z 353.476,A -85,B 0,C 180,E1 -15280.962,E2 -15280.962} C_VEL
LIN {X 0,Y 319.739,Z 353.471,A -85,B 0,C 180,E1 -15285.275,E2 -15285.275} C_VEL
LIN {X 0,Y 319.722,Z 353.473,A -85,B 0,C 180,E1 -15288.589,E2 -15288.589} C_VEL
LIN {X 0,Y 319.886,Z 353.452,A -85,B 0,C 180,E1 -15292.424,E2 -15292.424} C_VEL
LIN {X 0,Y 319.738,Z 353.471,A -85,B 0,C 180,E1 -15294.955,E2 -15294.955} C_VEL
LIN {X 0,Y 319.991,Z 353.44,A -85,B 0,C 180,E1 -15297.481,E2 -15297.481} C_VEL
LIN {X 0,Y 320.138,Z 353.422,A -85,B 0,C 180,E1 -15299.999,E2 -15299.999} C_VEL
LIN {X 0,Y 319.994,Z 353.439,A -85,B 0,C 180,E1 -15302.516,E2 -15302.516} C_VEL
LIN {X 0,Y 319.919,Z 353.448,A -85,B 0,C 180,E1 -15306.58,E2 -15306.58} C_VEL
LIN {X 0,Y 319.74,Z 353.471,A -85,B 0,C 180,E1 -15310.126,E2 -15310.126} C_VEL
LIN {X 0,Y 319.733,Z 353.475,A -85,B 0,C 180,E1 -15313.991,E2 -15313.991} C_VEL
LIN {X 0,Y 319.535,Z 353.502,A -85,B 0,C 180,E1 -15316.613,E2 -15316.613} C_VEL
LIN {X 0,Y 319.484,Z 354.11,A -85,B 0,C 180,E1 -15317.935,E2 -15317.935} C_VEL
LIN {X 0,Y 319.356,Z 356.326,A -85,B 0,C 180,E1 -15320.615,E2 -15320.615} C_VEL
LIN {X 0,Y 319.134,Z 358.676,A -85,B 0,C 180,E1 -15323.352,E2 -15323.352} C_VEL
LIN {X 0,Y 318.921,Z 361.16,A -85,B 0,C 180,E1 -15326.149,E2 -15326.149} C_VEL
LIN {X 0,Y 318.721,Z 363.794,A -85,B 0,C 180,E1 -15329.018,E2 -15329.018} C_VEL
LIN {X 0,Y 318.574,Z 365.811,A -85,B 0,C 180,E1 -15331.2,E2 -15331.2} C_VEL
LIN {X 0,Y 321.487,Z 376.108,A -85,B 0,C 180,E1 -15332.012,E2 -15332.012} C_VEL
LIN {X 0,Y 323.536,Z 385.408,A -85,B 0,C 180,E1 -15332.89,E2 -15332.89} C_VEL
LIN {X 0,Y 324.715,Z 393.099,A -85,B 0,C 180,E1 -15333.73,E2 -15333.73} C_VEL
LIN {X 0,Y 323.996,Z 400.646,A -85,B 0,C 180,E1 -15334.584,E2 -15334.584} C_VEL
LIN {X 0,Y 323.038,Z 408.119,A -85,B 0,C 180,E1 -15335.606,E2 -15335.606} C_VEL
LIN {X 0,Y 322.188,Z 414.915,A -85,B 0,C 180,E1 -15336.738,E2 -15336.738} C_VEL
LIN {X 0,Y 321.273,Z 421.376,A -85,B 0,C 180,E1 -15338.044,E2 -15338.044} C_VEL
LIN {X 0,Y 320.423,Z 427.226,A -85,B 0,C 180,E1 -15339.497,E2 -15339.497} C_VEL
LIN {X 0,Y 319.669,Z 432.07,A -85,B 0,C 180,E1 -15340.992,E2 -15340.992} C_VEL
LIN {X 0,Y 319.133,Z 435.66,A -85,B 0,C 180,E1 -15342.386,E2 -15342.386} C_VEL
LIN {X 0,Y 318.582,Z 439.193,A -85,B 0,C 180,E1 -15344.181,E2 -15344.181} C_VEL
LIN {X 0,Y 318.362,Z 440.464,A -85,B 0,C 180,E1 -15345.054,E2 -15345.054} C_VEL
LIN {X 0,Y 317.989,Z 442.297,A -85,B 0,C 180,E1 -15346.829,E2 -15346.829} C_VEL
LIN {X 0,Y 317.75,Z 443.172,A -85,B 0,C 180,E1 -15348.762,E2 -15348.762} C_VEL
LIN {X 0,Y 317.719,Z 442.9,A -85,B 0,C 180,E1 -15350.73,E2 -15350.73} C_VEL
LIN {X 0,Y 317.843,Z 441.332,A -85,B 0,C 180,E1 -15352.748,E2 -15352.748} C_VEL
LIN {X 0,Y 318.06,Z 439.491,A -85,B 0,C 180,E1 -15354.134,E2 -15354.134} C_VEL
LIN {X 0,Y 318.306,Z 436.523,A -85,B 0,C 180,E1 -15355.733,E2 -15355.733} C_VEL
LIN {X 0,Y 318.765,Z 432.013,A -85,B 0,C 180,E1 -15357.51,E2 -15357.51} C_VEL
LIN {X 0,Y 319.278,Z 426.653,A -85,B 0,C 180,E1 -15359.142,E2 -15359.142} C_VEL
LIN {X 0,Y 319.803,Z 421.739,A -85,B 0,C 180,E1 -15360.364,E2 -15360.364} C_VEL
LIN {X 0,Y 320.396,Z 415.68,A -85,B 0,C 180,E1 -15361.617,E2 -15361.617} C_VEL
LIN {X 0,Y 321.121,Z 408.108,A -85,B 0,C 180,E1 -15362.901,E2 -15362.901} C_VEL
LIN {X 0,Y 321.755,Z 401.162,A -85,B 0,C 180,E1 -15363.871,E2 -15363.871} C_VEL
LIN {X 0,Y 322.456,Z 392.629,A -85,B 0,C 180,E1 -15364.847,E2 -15364.847} C_VEL
LIN {X 0,Y 322.439,Z 387.415,A -85,B 0,C 180,E1 -15365.362,E2 -15365.362} C_VEL
LIN {X 0,Y 321.079,Z 378.928,A -85,B 0,C 180,E1 -15366.111,E2 -15366.111} C_VEL
LIN {X 0,Y 319.244,Z 369.365,A -85,B 0,C 180,E1 -15366.783,E2 -15366.783} C_VEL
LIN {X 0,Y 318.228,Z 364.333,A -85,B 0,C 180,E1 -15367.091,E2 -15367.091} C_VEL
LIN {X 0,Y 318.449,Z 359.641,A -85,B 0,C 180,E1 -15371.614,E2 -15371.614} C_VEL
LIN {X 0,Y 318.632,Z 356.555,A -85,B 0,C 180,E1 -15374.65,E2 -15374.65} C_VEL
LIN {X 0,Y 318.83,Z 353.93,A -85,B 0,C 180,E1 -15377.264,E2 -15377.264} C_VEL
LIN {X 0,Y 319.214,Z 353.533,A -85,B 0,C 180,E1 -15379.854,E2 -15379.854} C_VEL
LIN {X 0,Y 319.726,Z 353.473,A -85,B 0,C 180,E1 -15382.42,E2 -15382.42} C_VEL
LIN {X 0,Y 319.864,Z 353.452,A -85,B 0,C 180,E1 -15383.691,E2 -15383.691} C_VEL
LIN {X 0,Y 319.982,Z 353.437,A -85,B 0,C 180,E1 -15387.481,E2 -15387.481} C_VEL
LIN {X 0,Y 320.14,Z 353.421,A -85,B 0,C 180,E1 -15389.998,E2 -15389.998} C_VEL
LIN {X 0,Y 319.983,Z 353.438,A -85,B 0,C 180,E1 -15392.516,E2 -15392.516} C_VEL
LIN {X 0,Y 319.944,Z 353.443,A -85,B 0,C 180,E1 -15396.304,E2 -15396.304} C_VEL
LIN {X 0,Y 319.832,Z 353.455,A -85,B 0,C 180,E1 -15398.847,E2 -15398.847} C_VEL
LIN {X 0,Y 319.673,Z 353.475,A -85,B 0,C 180,E1 -15402.698,E2 -15402.698} C_VEL
LIN {X 0,Y 319.687,Z 353.474,A -85,B 0,C 180,E1 -15405.294,E2 -15405.294} C_VEL
LIN {X 0,Y 319.661,Z 353.478,A -85,B 0,C 180,E1 -15409.254,E2 -15409.254} C_VEL
LIN {X 0,Y 319.557,Z 353.492,A -85,B 0,C 180,E1 -15413.318,E2 -15413.318} C_VEL
LIN {X 0,Y 319.622,Z 353.482,A -85,B 0,C 180,E1 -15416.087,E2 -15416.087} C_VEL
LIN {X 0,Y 319.576,Z 353.488,A -85,B 0,C 180,E1 -15418.933,E2 -15418.933} C_VEL
LIN {X 0,Y 319.518,Z 353.495,A -85,B 0,C 180,E1 -15421.861,E2 -15421.861} C_VEL
LIN {X 0,Y 319.567,Z 353.491,A -85,B 0,C 180,E1 -15425.543,E2 -15425.543} C_VEL
LIN {X 0,Y 319.588,Z 353.485,A -85,B 0,C 180,E1 -15428.003,E2 -15428.003} C_VEL
LIN {X 0,Y 319.587,Z 353.487,A -85,B 0,C 180,E1 -15431.612,E2 -15431.612} C_VEL
LIN {X 0,Y 319.631,Z 353.483,A -85,B 0,C 180,E1 -15435.285,E2 -15435.285} C_VEL
LIN {X 0,Y 319.569,Z 353.491,A -85,B 0,C 180,E1 -15438.72,E2 -15438.72} C_VEL
LIN {X 0,Y 319.585,Z 353.487,A -85,B 0,C 180,E1 -15442.339,E2 -15442.339} C_VEL
LIN {X 0,Y 319.546,Z 353.493,A -85,B 0,C 180,E1 -15445.124,E2 -15445.124} C_VEL
LIN {X 0,Y 319.556,Z 353.491,A -85,B 0,C 180,E1 -15449.058,E2 -15449.058} C_VEL
LIN {X 0,Y 319.596,Z 353.489,A -85,B 0,C 180,E1 -15452.499,E2 -15452.499} C_VEL
LIN {X 0,Y 319.613,Z 353.482,A -85,B 0,C 180,E1 -15455.306,E2 -15455.306} C_VEL
LIN {X 0,Y 319.628,Z 353.482,A -85,B 0,C 180,E1 -15458.052,E2 -15458.052} C_VEL
LIN {X 0,Y 319.64,Z 353.478,A -85,B 0,C 180,E1 -15460.276,E2 -15460.276} C_VEL
LIN {X 0,Y 319.041,Z 353.557,A -85,B 0,C 180,E1 -15461.327,E2 -15461.327} C_VEL
LIN {X 0,Y 316.268,Z 353.907,A -85,B 0,C 180,E1 -15463.039,E2 -15463.039} C_VEL
LIN {X 0,Y 313.855,Z 354.206,A -85,B 0,C 180,E1 -15464.426,E2 -15464.426} C_VEL
LIN {X 0,Y 312.775,Z 354.336,A -85,B 0,C 180,E1 -15465.499,E2 -15465.499} C_VEL
LIN {X 0,Y 312.664,Z 354.347,A -85,B 0,C 180,E1 -15465.862,E2 -15465.862} C_VEL
LIN {X 0,Y 312.692,Z 354.345,A -85,B 0,C 180,E1 -15469.643,E2 -15469.643} C_VEL
LIN {X 0,Y 312.86,Z 354.328,A -85,B 0,C 180,E1 -15472.255,E2 -15472.255} C_VEL
LIN {X 0,Y 312.707,Z 354.342,A -85,B 0,C 180,E1 -15474.844,E2 -15474.844} C_VEL
LIN {X 0,Y 312.98,Z 354.309,A -85,B 0,C 180,E1 -15478.715,E2 -15478.715} C_VEL
LIN {X 0,Y 312.982,Z 354.309,A -85,B 0,C 180,E1 -15481.288,E2 -15481.288} C_VEL
LIN {X 0,Y 312.71,Z 354.342,A -85,B 0,C 180,E1 -15485.159,E2 -15485.159} C_VEL
LIN {X 0,Y 312.862,Z 354.328,A -85,B 0,C 180,E1 -15487.747,E2 -15487.747} C_VEL
LIN {X 0,Y 312.663,Z 354.353,A -85,B 0,C 180,E1 -15491.673,E2 -15491.673} C_VEL
LIN {X 0,Y 312.691,Z 354.345,A -85,B 0,C 180,E1 -15494.889,E2 -15494.889} C_VEL
LIN {X 0,Y 312.621,Z 354.356,A -85,B 0,C 180,E1 -15499.238,E2 -15499.238} C_VEL
LIN {X 0,Y 312.538,Z 354.364,A -85,B 0,C 180,E1 -15502.791,E2 -15502.791} C_VEL
LIN {X 0,Y 312.595,Z 354.357,A -85,B 0,C 180,E1 -15505.937,E2 -15505.937} C_VEL
LIN {X 0,Y 312.538,Z 354.365,A -85,B 0,C 180,E1 -15509.652,E2 -15509.652} C_VEL
LIN {X 0,Y 312.513,Z 354.368,A -85,B 0,C 180,E1 -15513.691,E2 -15513.691} C_VEL
LIN {X 0,Y 312.514,Z 354.369,A -85,B 0,C 180,E1 -15517.388,E2 -15517.388} C_VEL
LIN {X 0,Y 312.485,Z 354.373,A -85,B 0,C 180,E1 -15520.711,E2 -15520.711} C_VEL
LIN {X 0,Y 312.468,Z 354.373,A -85,B 0,C 180,E1 -15524.208,E2 -15524.208} C_VEL
LIN {X 0,Y 312.508,Z 354.368,A -85,B 0,C 180,E1 -15527.915,E2 -15527.915} C_VEL
LIN {X 0,Y 312.601,Z 354.518,A -85,B 0,C 180,E1 -15529.311,E2 -15529.311} C_VEL
LIN {X 0,Y 313.469,Z 359.393,A -85,B 0,C 180,E1 -15532.749,E2 -15532.749} C_VEL
LIN {X 0,Y 314.183,Z 364.209,A -85,B 0,C 180,E1 -15536,E2 -15536} C_VEL
LIN {X 0,Y 313.811,Z 367.91,A -85,B 0,C 180,E1 -15538.326,E2 -15538.326} C_VEL
LIN {X 0,Y 313.003,Z 373.673,A -85,B 0,C 180,E1 -15541.869,E2 -15541.869} C_VEL
LIN {X 0,Y 312.29,Z 379.548,A -85,B 0,C 180,E1 -15545.399,E2 -15545.399} C_VEL
LIN {X 0,Y 311.746,Z 385.396,A -85,B 0,C 180,E1 -15548.859,E2 -15548.859} C_VEL
LIN {X 0,Y 311.265,Z 391.759,A -85,B 0,C 180,E1 -15552.552,E2 -15552.552} C_VEL
LIN {X 0,Y 312.688,Z 404.391,A -85,B 0,C 180,E1 -15553.29,E2 -15553.29} C_VEL
LIN {X 0,Y 313.521,Z 412.992,A -85,B 0,C 180,E1 -15553.962,E2 -15553.962} C_VEL
LIN {X 0,Y 314.14,Z 423.079,A -85,B 0,C 180,E1 -15554.961,E2 -15554.961} C_VEL
LIN {X 0,Y 314.117,Z 429.761,A -85,B 0,C 180,E1 -15555.754,E2 -15555.754} C_VEL
LIN {X 0,Y 313.245,Z 437.693,A -85,B 0,C 180,E1 -15556.872,E2 -15556.872} C_VEL
LIN {X 0,Y 312.629,Z 444.282,A -85,B 0,C 180,E1 -15558,E2 -15558} C_VEL
LIN {X 0,Y 312.012,Z 450.55,A -85,B 0,C 180,E1 -15559.292,E2 -15559.292} C_VEL
LIN {X 0,Y 311.563,Z 455.759,A -85,B 0,C 180,E1 -15560.589,E2 -15560.589} C_VEL
LIN {X 0,Y 311.131,Z 461.053,A -85,B 0,C 180,E1 -15562.212,E2 -15562.212} C_VEL
LIN {X 0,Y 310.907,Z 464.447,A -85,B 0,C 180,E1 -15563.512,E2 -15563.512} C_VEL
LIN {X 0,Y 310.792,Z 467.206,A -85,B 0,C 180,E1 -15564.812,E2 -15564.812} C_VEL
LIN {X 0,Y 310.85,Z 469.395,A -85,B 0,C 180,E1 -15566.113,E2 -15566.113} C_VEL
LIN {X 0,Y 310.771,Z 470.991,A -85,B 0,C 180,E1 -15567.409,E2 -15567.409} C_VEL
LIN {X 0,Y 310.793,Z 471.984,A -85,B 0,C 180,E1 -15568.706,E2 -15568.706} C_VEL
LIN {X 0,Y 310.856,Z 472.488,A -85,B 0,C 180,E1 -15570.002,E2 -15570.002} C_VEL
LIN {X 0,Y 310.775,Z 472.511,A -85,B 0,C 180,E1 -15571.297,E2 -15571.297} C_VEL
LIN {X 0,Y 310.747,Z 472.063,A -85,B 0,C 180,E1 -15572.594,E2 -15572.594} C_VEL
LIN {X 0,Y 310.784,Z 471.035,A -85,B 0,C 180,E1 -15573.892,E2 -15573.892} C_VEL
LIN {X 0,Y 310.788,Z 468.729,A -85,B 0,C 180,E1 -15575.731,E2 -15575.731} C_VEL
LIN {X 0,Y 311.182,Z 464.735,A -85,B 0,C 180,E1 -15577.79,E2 -15577.79} C_VEL
LIN {X 0,Y 311.76,Z 459.542,A -85,B 0,C 180,E1 -15579.735,E2 -15579.735} C_VEL
LIN {X 0,Y 312.488,Z 453.996,A -85,B 0,C 180,E1 -15581.351,E2 -15581.351} C_VEL
LIN {X 0,Y 313.471,Z 447.117,A -85,B 0,C 180,E1 -15582.957,E2 -15582.957} C_VEL
LIN {X 0,Y 314.721,Z 438.301,A -85,B 0,C 180,E1 -15584.551,E2 -15584.551} C_VEL
LIN {X 0,Y 315.589,Z 431.918,A -85,B 0,C 180,E1 -15585.501,E2 -15585.501} C_VEL
LIN {X 0,Y 315.835,Z 423.946,A -85,B 0,C 180,E1 -15586.526,E2 -15586.526} C_VEL
LIN {X 0,Y 315.456,Z 414.936,A -85,B 0,C 180,E1 -15587.504,E2 -15587.504} C_VEL
LIN {X 0,Y 314.5,Z 405.856,A -85,B 0,C 180,E1 -15588.333,E2 -15588.333} C_VEL
LIN {X 0,Y 312.845,Z 396.165,A -85,B 0,C 180,E1 -15589.071,E2 -15589.071} C_VEL
LIN {X 0,Y 311.602,Z 390.281,A -85,B 0,C 180,E1 -15589.455,E2 -15589.455} C_VEL
LIN {X 0,Y 312.192,Z 384.016,A -85,B 0,C 180,E1 -15593.202,E2 -15593.202} C_VEL
LIN {X 0,Y 313.074,Z 377.223,A -85,B 0,C 180,E1 -15597.401,E2 -15597.401} C_VEL
LIN {X 0,Y 314.243,Z 370.453,A -85,B 0,C 180,E1 -15601.802,E2 -15601.802} C_VEL
LIN {X 0,Y 314.555,Z 366.912,A -85,B 0,C 180,E1 -15604.24,E2 -15604.24} C_VEL
LIN {X 0,Y 313.996,Z 363.049,A -85,B 0,C 180,E1 -15607.182,E2 -15607.182} C_VEL
LIN {X 0,Y 313.366,Z 358.963,A -85,B 0,C 180,E1 -15610.573,E2 -15610.573} C_VEL
LIN {X 0,Y 312.578,Z 355.014,A -85,B 0,C 180,E1 -15614.189,E2 -15614.189} C_VEL
LIN {X 0,Y 312.451,Z 354.385,A -85,B 0,C 180,E1 -15614.983,E2 -15614.983} C_VEL
LIN {X 0,Y 312.492,Z 354.374,A -85,B 0,C 180,E1 -15617.919,E2 -15617.919} C_VEL
LIN {X 0,Y 312.513,Z 354.371,A -85,B 0,C 180,E1 -15621.918,E2 -15621.918} C_VEL
LIN {X 0,Y 312.54,Z 354.368,A -85,B 0,C 180,E1 -15624.22,E2 -15624.22} C_VEL
LIN {X 0,Y 312.512,Z 354.371,A -85,B 0,C 180,E1 -15627.334,E2 -15627.334} C_VEL
LIN {X 0,Y 312.552,Z 354.365,A -85,B 0,C 180,E1 -15631.279,E2 -15631.279} C_VEL
LIN {X 0,Y 312.594,Z 354.361,A -85,B 0,C 180,E1 -15634.711,E2 -15634.711} C_VEL
LIN {X 0,Y 312.596,Z 354.361,A -85,B 0,C 180,E1 -15637.529,E2 -15637.529} C_VEL
LIN {X 0,Y 312.646,Z 354.354,A -85,B 0,C 180,E1 -15641.656,E2 -15641.656} C_VEL
LIN {X 0,Y 312.702,Z 354.348,A -85,B 0,C 180,E1 -15645.685,E2 -15645.685} C_VEL
LIN {X 0,Y 312.693,Z 354.349,A -85,B 0,C 180,E1 -15649.64,E2 -15649.64} C_VEL
LIN {X 0,Y 312.824,Z 354.331,A -85,B 0,C 180,E1 -15652.252,E2 -15652.252} C_VEL
LIN {X 0,Y 312.707,Z 354.347,A -85,B 0,C 180,E1 -15654.841,E2 -15654.841} C_VEL
LIN {X 0,Y 312.994,Z 354.307,A -85,B 0,C 180,E1 -15658.712,E2 -15658.712} C_VEL
LIN {X 0,Y 312.995,Z 354.308,A -85,B 0,C 180,E1 -15661.285,E2 -15661.285} C_VEL
LIN {X 0,Y 312.717,Z 354.344,A -85,B 0,C 180,E1 -15665.156,E2 -15665.156} C_VEL
LIN {X 0,Y 312.886,Z 354.325,A -85,B 0,C 180,E1 -15666.557,E2 -15666.557} C_VEL
LIN {X 0,Y 312.69,Z 354.349,A -85,B 0,C 180,E1 -15670.357,E2 -15670.357} C_VEL
LIN {X 0,Y 312.685,Z 354.354,A -85,B 0,C 180,E1 -15674.313,E2 -15674.313} C_VEL
LIN {X 0,Y 312.463,Z 354.521,A -85,B 0,C 180,E1 -15677,E2 -15677} C_VEL
LIN {X 0,Y 312.39,Z 356.672,A -85,B 0,C 180,E1 -15679.721,E2 -15679.721} C_VEL
LIN {X 0,Y 312.173,Z 359.063,A -85,B 0,C 180,E1 -15682.622,E2 -15682.622} C_VEL
LIN {X 0,Y 311.954,Z 361.718,A -85,B 0,C 180,E1 -15685.687,E2 -15685.687} C_VEL
LIN {X 0,Y 311.626,Z 365.374,A -85,B 0,C 180,E1 -15689.744,E2 -15689.744} C_VEL
LIN {X 0,Y 311.582,Z 366.189,A -85,B 0,C 180,E1 -15690.637,E2 -15690.637} C_VEL
LIN {X 0,Y 314.884,Z 377.846,A -85,B 0,C 180,E1 -15691.633,E2 -15691.633} C_VEL
LIN {X 0,Y 316.648,Z 385.651,A -85,B 0,C 180,E1 -15692.4,E2 -15692.4} C_VEL
LIN {X 0,Y 317.948,Z 394.075,A -85,B 0,C 180,E1 -15693.354,E2 -15693.354} C_VEL
LIN {X 0,Y 317.058,Z 402.942,A -85,B 0,C 180,E1 -15694.417,E2 -15694.417} C_VEL
LIN {X 0,Y 315.837,Z 411.835,A -85,B 0,C 180,E1 -15695.738,E2 -15695.738} C_VEL
LIN {X 0,Y 314.774,Z 419.727,A -85,B 0,C 180,E1 -15697.239,E2 -15697.239} C_VEL
LIN {X 0,Y 313.712,Z 426.368,A -85,B 0,C 180,E1 -15698.847,E2 -15698.847} C_VEL
LIN {X 0,Y 313.006,Z 431.007,A -85,B 0,C 180,E1 -15700.232,E2 -15700.232} C_VEL
LIN {X 0,Y 312.43,Z 434.153,A -85,B 0,C 180,E1 -15701.334,E2 -15701.334} C_VEL
LIN {X 0,Y 311.802,Z 438.122,A -85,B 0,C 180,E1 -15703.159,E2 -15703.159} C_VEL
LIN {X 0,Y 311.445,Z 440.214,A -85,B 0,C 180,E1 -15704.388,E2 -15704.388} C_VEL
LIN {X 0,Y 310.999,Z 442.378,A -85,B 0,C 180,E1 -15706.312,E2 -15706.312} C_VEL
LIN {X 0,Y 310.692,Z 443.434,A -85,B 0,C 180,E1 -15708.283,E2 -15708.283} C_VEL
LIN {X 0,Y 310.618,Z 443.348,A -85,B 0,C 180,E1 -15710.286,E2 -15710.286} C_VEL
LIN {X 0,Y 310.733,Z 442.044,A -85,B 0,C 180,E1 -15712.36,E2 -15712.36} C_VEL
LIN {X 0,Y 311.015,Z 439.343,A -85,B 0,C 180,E1 -15714.435,E2 -15714.435} C_VEL
LIN {X 0,Y 311.334,Z 435.965,A -85,B 0,C 180,E1 -15716.167,E2 -15716.167} C_VEL
LIN {X 0,Y 311.718,Z 432.282,A -85,B 0,C 180,E1 -15717.623,E2 -15717.623} C_VEL
LIN {X 0,Y 312.21,Z 427.153,A -85,B 0,C 180,E1 -15719.224,E2 -15719.224} C_VEL
LIN {X 0,Y 312.725,Z 422.741,A -85,B 0,C 180,E1 -15720.367,E2 -15720.367} C_VEL
LIN {X 0,Y 313.433,Z 415.439,A -85,B 0,C 180,E1 -15721.907,E2 -15721.907} C_VEL
LIN {X 0,Y 314.102,Z 408.782,A -85,B 0,C 180,E1 -15723.057,E2 -15723.057} C_VEL
LIN {X 0,Y 314.855,Z 400.77,A -85,B 0,C 180,E1 -15724.196,E2 -15724.196} C_VEL
LIN {X 0,Y 315.652,Z 390.884,A -85,B 0,C 180,E1 -15725.323,E2 -15725.323} C_VEL
LIN {X 0,Y 314.331,Z 380.951,A -85,B 0,C 180,E1 -15726.267,E2 -15726.267} C_VEL
LIN {X 0,Y 312.254,Z 370.098,A -85,B 0,C 180,E1 -15727.065,E2 -15727.065} C_VEL
LIN {X 0,Y 311.165,Z 364.629,A -85,B 0,C 180,E1 -15727.419,E2 -15727.419} C_VEL
LIN {X 0,Y 311.379,Z 360.388,A -85,B 0,C 180,E1 -15731.578,E2 -15731.578} C_VEL
LIN {X 0,Y 311.66,Z 356.117,A -85,B 0,C 180,E1 -15735.842,E2 -15735.842} C_VEL
LIN {X 0,Y 311.749,Z 355.011,A -85,B 0,C 180,E1 -15736.97,E2 -15736.97} C_VEL
LIN {X 0,Y 311.888,Z 354.449,A -85,B 0,C 180,E1 -15738.297,E2 -15738.297} C_VEL
LIN {X 0,Y 312.654,Z 354.354,A -85,B 0,C 180,E1 -15742.247,E2 -15742.247} C_VEL
LIN {X 0,Y 312.794,Z 354.332,A -85,B 0,C 180,E1 -15743.548,E2 -15743.548} C_VEL
LIN {X 0,Y 312.928,Z 354.315,A -85,B 0,C 180,E1 -15747.424,E2 -15747.424} C_VEL
LIN {X 0,Y 313.093,Z 354.299,A -85,B 0,C 180,E1 -15749.998,E2 -15749.998} C_VEL
LIN {X 0,Y 312.929,Z 354.316,A -85,B 0,C 180,E1 -15752.573,E2 -15752.573} C_VEL
LIN {X 0,Y 312.902,Z 354.32,A -85,B 0,C 180,E1 -15756.446,E2 -15756.446} C_VEL
LIN {X 0,Y 312.777,Z 354.334,A -85,B 0,C 180,E1 -15759.048,E2 -15759.048} C_VEL
LIN {X 0,Y 312.625,Z 354.353,A -85,B 0,C 180,E1 -15762.99,E2 -15762.99} C_VEL
LIN {X 0,Y 312.626,Z 354.357,A -85,B 0,C 180,E1 -15765.648,E2 -15765.648} C_VEL
LIN {X 0,Y 312.617,Z 354.355,A -85,B 0,C 180,E1 -15769.235,E2 -15769.235} C_VEL
LIN {X 0,Y 312.533,Z 354.364,A -85,B 0,C 180,E1 -15772.788,E2 -15772.788} C_VEL
LIN {X 0,Y 312.59,Z 354.359,A -85,B 0,C 180,E1 -15775.935,E2 -15775.935} C_VEL
LIN {X 0,Y 312.532,Z 354.367,A -85,B 0,C 180,E1 -15779.649,E2 -15779.649} C_VEL
LIN {X 0,Y 312.505,Z 354.37,A -85,B 0,C 180,E1 -15783.688,E2 -15783.688} C_VEL
LIN {X 0,Y 312.541,Z 354.367,A -85,B 0,C 180,E1 -15787.381,E2 -15787.381} C_VEL
LIN {X 0,Y 312.521,Z 354.367,A -85,B 0,C 180,E1 -15790.702,E2 -15790.702} C_VEL
LIN {X 0,Y 312.581,Z 354.358,A -85,B 0,C 180,E1 -15794.184,E2 -15794.184} C_VEL
LIN {X 0,Y 312.542,Z 354.363,A -85,B 0,C 180,E1 -15797.904,E2 -15797.904} C_VEL
LIN {X 0,Y 312.544,Z 354.362,A -85,B 0,C 180,E1 -15801.905,E2 -15801.905} C_VEL
LIN {X 0,Y 312.492,Z 354.369,A -85,B 0,C 180,E1 -15805.79,E2 -15805.79} C_VEL
LIN {X 0,Y 312.51,Z 354.371,A -85,B 0,C 180,E1 -15808.854,E2 -15808.854} C_VEL
LIN {X 0,Y 312.561,Z 354.36,A -85,B 0,C 180,E1 -15811.825,E2 -15811.825} C_VEL
LIN {X 0,Y 312.581,Z 354.362,A -85,B 0,C 180,E1 -15814.712,E2 -15814.712} C_VEL
LIN {X 0,Y 312.608,Z 354.355,A -85,B 0,C 180,E1 -15817.532,E2 -15817.532} C_VEL
LIN {X 0,Y 312.632,Z 354.352,A -85,B 0,C 180,E1 -15821.658,E2 -15821.658} C_VEL
LIN {X 0,Y 312.664,Z 354.347,A -85,B 0,C 180,E1 -15825.862,E2 -15825.862} C_VEL
LIN {X 0,Y 311.954,Z 354.437,A -85,B 0,C 180,E1 -15826.937,E2 -15826.937} C_VEL
LIN {X 0,Y 309.158,Z 354.786,A -85,B 0,C 180,E1 -15828.689,E2 -15828.689} C_VEL
LIN {X 0,Y 306.835,Z 355.078,A -85,B 0,C 180,E1 -15830.11,E2 -15830.11} C_VEL
LIN {X 0,Y 305.856,Z 355.196,A -85,B 0,C 180,E1 -15831.208,E2 -15831.208} C_VEL
LIN {X 0,Y 305.783,Z 355.206,A -85,B 0,C 180,E1 -15831.579,E2 -15831.579} C_VEL
LIN {X 0,Y 305.841,Z 355.198,A -85,B 0,C 180,E1 -15833.404,E2 -15833.404} C_VEL
LIN {X 0,Y 305.946,Z 355.185,A -85,B 0,C 180,E1 -15838.685,E2 -15838.685} C_VEL
LIN {X 0,Y 305.949,Z 355.185,A -85,B 0,C 180,E1 -15841.318,E2 -15841.318} C_VEL
LIN {X 0,Y 305.842,Z 355.198,A -85,B 0,C 180,E1 -15846.599,E2 -15846.599} C_VEL
LIN {X 0,Y 305.726,Z 355.214,A -85,B 0,C 180,E1 -15849.261,E2 -15849.261} C_VEL
LIN {X 0,Y 305.582,Z 355.232,A -85,B 0,C 180,E1 -15853.298,E2 -15853.298} C_VEL
LIN {X 0,Y 305.585,Z 355.231,A -85,B 0,C 180,E1 -15856.022,E2 -15856.022} C_VEL
LIN {X 0,Y 305.568,Z 355.237,A -85,B 0,C 180,E1 -15859.446,E2 -15859.446} C_VEL
LIN {X 0,Y 305.483,Z 355.244,A -85,B 0,C 180,E1 -15863.043,E2 -15863.043} C_VEL
LIN {X 0,Y 305.54,Z 355.235,A -85,B 0,C 180,E1 -15866.229,E2 -15866.229} C_VEL
LIN {X 0,Y 305.489,Z 355.245,A -85,B 0,C 180,E1 -15869.052,E2 -15869.052} C_VEL
LIN {X 0,Y 305.459,Z 355.248,A -85,B 0,C 180,E1 -15873.519,E2 -15873.519} C_VEL
LIN {X 0,Y 305.466,Z 355.247,A -85,B 0,C 180,E1 -15876.742,E2 -15876.742} C_VEL
LIN {X 0,Y 305.449,Z 355.249,A -85,B 0,C 180,E1 -15880.602,E2 -15880.602} C_VEL
LIN {X 0,Y 305.414,Z 355.253,A -85,B 0,C 180,E1 -15884.495,E2 -15884.495} C_VEL
LIN {X 0,Y 305.465,Z 355.246,A -85,B 0,C 180,E1 -15888.15,E2 -15888.15} C_VEL
LIN {X 0,Y 305.543,Z 355.456,A -85,B 0,C 180,E1 -15889.15,E2 -15889.15} C_VEL
LIN {X 0,Y 306.409,Z 360.174,A -85,B 0,C 180,E1 -15892.571,E2 -15892.571} C_VEL
LIN {X 0,Y 307.05,Z 364.381,A -85,B 0,C 180,E1 -15895.488,E2 -15895.488} C_VEL
LIN {X 0,Y 307.121,Z 366.194,A -85,B 0,C 180,E1 -15896.69,E2 -15896.69} C_VEL
LIN {X 0,Y 306.435,Z 370.911,A -85,B 0,C 180,E1 -15899.7,E2 -15899.7} C_VEL
LIN {X 0,Y 305.469,Z 377.968,A -85,B 0,C 180,E1 -15904.081,E2 -15904.081} C_VEL
LIN {X 0,Y 304.742,Z 384.967,A -85,B 0,C 180,E1 -15908.348,E2 -15908.348} C_VEL
LIN {X 0,Y 304.208,Z 391.438,A -85,B 0,C 180,E1 -15912.223,E2 -15912.223} C_VEL
LIN {X 0,Y 305.695,Z 404.893,A -85,B 0,C 180,E1 -15913.043,E2 -15913.043} C_VEL
LIN {X 0,Y 306.615,Z 414.743,A -85,B 0,C 180,E1 -15913.866,E2 -15913.866} C_VEL
LIN {X 0,Y 307.082,Z 422.819,A -85,B 0,C 180,E1 -15914.701,E2 -15914.701} C_VEL
LIN {X 0,Y 307.197,Z 428.82,A -85,B 0,C 180,E1 -15915.426,E2 -15915.426} C_VEL
LIN {X 0,Y 306.332,Z 436.858,A -85,B 0,C 180,E1 -15916.57,E2 -15916.57} C_VEL
LIN {X 0,Y 305.652,Z 443.525,A -85,B 0,C 180,E1 -15917.722,E2 -15917.722} C_VEL
LIN {X 0,Y 304.996,Z 449.862,A -85,B 0,C 180,E1 -15919.043,E2 -15919.043} C_VEL
LIN {X 0,Y 304.539,Z 455.134,A -85,B 0,C 180,E1 -15920.37,E2 -15920.37} C_VEL
LIN {X 0,Y 304.073,Z 460.481,A -85,B 0,C 180,E1 -15922.03,E2 -15922.03} C_VEL
LIN {X 0,Y 303.787,Z 464.952,A -85,B 0,C 180,E1 -15923.809,E2 -15923.809} C_VEL
LIN {X 0,Y 303.757,Z 468.959,A -85,B 0,C 180,E1 -15926.022,E2 -15926.022} C_VEL
LIN {X 0,Y 303.694,Z 470.565,A -85,B 0,C 180,E1 -15927.349,E2 -15927.349} C_VEL
LIN {X 0,Y 303.703,Z 471.59,A -85,B 0,C 180,E1 -15928.676,E2 -15928.676} C_VEL
LIN {X 0,Y 303.764,Z 472.132,A -85,B 0,C 180,E1 -15930.002,E2 -15930.002} C_VEL
LIN {X 0,Y 303.685,Z 472.193,A -85,B 0,C 180,E1 -15931.328,E2 -15931.328} C_VEL
LIN {X 0,Y 303.669,Z 471.771,A -85,B 0,C 180,E1 -15932.655,E2 -15932.655} C_VEL
LIN {X 0,Y 303.694,Z 470.752,A -85,B 0,C 180,E1 -15933.983,E2 -15933.983} C_VEL
LIN {X 0,Y 303.698,Z 468.74,A -85,B 0,C 180,E1 -15935.68,E2 -15935.68} C_VEL
LIN {X 0,Y 304.117,Z 464.573,A -85,B 0,C 180,E1 -15937.972,E2 -15937.972} C_VEL
LIN {X 0,Y 304.519,Z 461.384,A -85,B 0,C 180,E1 -15939.299,E2 -15939.299} C_VEL
LIN {X 0,Y 305.192,Z 456.336,A -85,B 0,C 180,E1 -15940.953,E2 -15940.953} C_VEL
LIN {X 0,Y 306.135,Z 450.026,A -85,B 0,C 180,E1 -15942.599,E2 -15942.599} C_VEL
LIN {X 0,Y 307.074,Z 443.891,A -85,B 0,C 180,E1 -15943.907,E2 -15943.907} C_VEL
LIN {X 0,Y 308.039,Z 437.492,A -85,B 0,C 180,E1 -15945.043,E2 -15945.043} C_VEL
LIN {X 0,Y 308.924,Z 430.337,A -85,B 0,C 180,E1 -15946.109,E2 -15946.109} C_VEL
LIN {X 0,Y 308.998,Z 421.859,A -85,B 0,C 180,E1 -15947.2,E2 -15947.2} C_VEL
LIN {X 0,Y 308.533,Z 413.802,A -85,B 0,C 180,E1 -15948.083,E2 -15948.083} C_VEL
LIN {X 0,Y 307.589,Z 405.48,A -85,B 0,C 180,E1 -15948.862,E2 -15948.862} C_VEL
LIN {X 0,Y 305.834,Z 395.564,A -85,B 0,C 180,E1 -15949.654,E2 -15949.654} C_VEL
LIN {X 0,Y 304.646,Z 389.84,A -85,B 0,C 180,E1 -15950.074,E2 -15950.074} C_VEL
LIN {X 0,Y 305.222,Z 383.874,A -85,B 0,C 180,E1 -15953.764,E2 -15953.764} C_VEL
LIN {X 0,Y 306.02,Z 378.236,A -85,B 0,C 180,E1 -15957.345,E2 -15957.345} C_VEL
LIN {X 0,Y 307.192,Z 371.641,A -85,B 0,C 180,E1 -15961.751,E2 -15961.751} C_VEL
LIN {X 0,Y 307.531,Z 369.456,A -85,B 0,C 180,E1 -15963.264,E2 -15963.264} C_VEL
LIN {X 0,Y 307.324,Z 366.251,A -85,B 0,C 180,E1 -15965.674,E2 -15965.674} C_VEL
LIN {X 0,Y 306.714,Z 362.403,A -85,B 0,C 180,E1 -15968.823,E2 -15968.823} C_VEL
LIN {X 0,Y 306.164,Z 359.063,A -85,B 0,C 180,E1 -15971.738,E2 -15971.738} C_VEL
LIN {X 0,Y 305.413,Z 355.261,A -85,B 0,C 180,E1 -15975.51,E2 -15975.51} C_VEL
LIN {X 0,Y 305.449,Z 355.252,A -85,B 0,C 180,E1 -15978.143,E2 -15978.143} C_VEL
LIN {X 0,Y 305.484,Z 355.247,A -85,B 0,C 180,E1 -15981.598,E2 -15981.598} C_VEL
LIN {X 0,Y 305.47,Z 355.248,A -85,B 0,C 180,E1 -15984.887,E2 -15984.887} C_VEL
LIN {X 0,Y 305.458,Z 355.249,A -85,B 0,C 180,E1 -15988.356,E2 -15988.356} C_VEL
LIN {X 0,Y 305.521,Z 355.241,A -85,B 0,C 180,E1 -15991.113,E2 -15991.113} C_VEL
LIN {X 0,Y 305.579,Z 355.234,A -85,B 0,C 180,E1 -15994.088,E2 -15994.088} C_VEL
LIN {X 0,Y 305.509,Z 355.242,A -85,B 0,C 180,E1 -15998.402,E2 -15998.402} C_VEL
LIN {X 0,Y 305.598,Z 355.232,A -85,B 0,C 180,E1 -16001.217,E2 -16001.217} C_VEL
LIN {X 0,Y 305.657,Z 355.225,A -85,B 0,C 180,E1 -16005.348,E2 -16005.348} C_VEL
LIN {X 0,Y 305.632,Z 355.228,A -85,B 0,C 180,E1 -16009.398,E2 -16009.398} C_VEL
LIN {X 0,Y 305.771,Z 355.21,A -85,B 0,C 180,E1 -16012.072,E2 -16012.072} C_VEL
LIN {X 0,Y 305.677,Z 355.222,A -85,B 0,C 180,E1 -16014.722,E2 -16014.722} C_VEL
LIN {X 0,Y 305.961,Z 355.183,A -85,B 0,C 180,E1 -16018.683,E2 -16018.683} C_VEL
LIN {X 0,Y 305.962,Z 355.184,A -85,B 0,C 180,E1 -16021.315,E2 -16021.315} C_VEL
LIN {X 0,Y 305.688,Z 355.22,A -85,B 0,C 180,E1 -16025.275,E2 -16025.275} C_VEL
LIN {X 0,Y 305.777,Z 355.21,A -85,B 0,C 180,E1 -16027.925,E2 -16027.925} C_VEL
LIN {X 0,Y 305.603,Z 355.232,A -85,B 0,C 180,E1 -16031.944,E2 -16031.944} C_VEL
LIN {X 0,Y 305.59,Z 355.238,A -85,B 0,C 180,E1 -16034.997,E2 -16034.997} C_VEL
LIN {X 0,Y 305.487,Z 355.253,A -85,B 0,C 180,E1 -16036.024,E2 -16036.024} C_VEL
LIN {X 0,Y 305.453,Z 357.04,A -85,B 0,C 180,E1 -16038.789,E2 -16038.789} C_VEL
LIN {X 0,Y 305.126,Z 360.34,A -85,B 0,C 180,E1 -16042.876,E2 -16042.876} C_VEL
LIN {X 0,Y 304.891,Z 362.963,A -85,B 0,C 180,E1 -16045.972,E2 -16045.972} C_VEL
LIN {X 0,Y 304.571,Z 366.575,A -85,B 0,C 180,E1 -16050.075,E2 -16050.075} C_VEL
LIN {X 0,Y 307.755,Z 377.398,A -85,B 0,C 180,E1 -16051.012,E2 -16051.012} C_VEL
LIN {X 0,Y 309.889,Z 386.611,A -85,B 0,C 180,E1 -16051.964,E2 -16051.964} C_VEL
LIN {X 0,Y 311.03,Z 394.121,A -85,B 0,C 180,E1 -16052.839,E2 -16052.839} C_VEL
LIN {X 0,Y 311.078,Z 397.847,A -85,B 0,C 180,E1 -16053.286,E2 -16053.286} C_VEL
LIN {X 0,Y 309.836,Z 407.328,A -85,B 0,C 180,E1 -16054.544,E2 -16054.544} C_VEL
LIN {X 0,Y 308.601,Z 415.804,A -85,B 0,C 180,E1 -16056.002,E2 -16056.002} C_VEL
LIN {X 0,Y 307.715,Z 421.479,A -85,B 0,C 180,E1 -16057.189,E2 -16057.189} C_VEL
LIN {X 0,Y 306.658,Z 427.793,A -85,B 0,C 180,E1 -16058.81,E2 -16058.81} C_VEL
LIN {X 0,Y 305.692,Z 433.444,A -85,B 0,C 180,E1 -16060.65,E2 -16060.65} C_VEL
LIN {X 0,Y 304.936,Z 437.699,A -85,B 0,C 180,E1 -16062.478,E2 -16062.478} C_VEL
LIN {X 0,Y 304.382,Z 440.715,A -85,B 0,C 180,E1 -16064.292,E2 -16064.292} C_VEL
LIN {X 0,Y 303.971,Z 442.677,A -85,B 0,C 180,E1 -16066.081,E2 -16066.081} C_VEL
LIN {X 0,Y 303.648,Z 443.708,A -85,B 0,C 180,E1 -16067.838,E2 -16067.838} C_VEL
LIN {X 0,Y 303.524,Z 443.796,A -85,B 0,C 180,E1 -16069.825,E2 -16069.825} C_VEL
LIN {X 0,Y 303.582,Z 442.705,A -85,B 0,C 180,E1 -16071.913,E2 -16071.913} C_VEL
LIN {X 0,Y 303.855,Z 440.329,A -85,B 0,C 180,E1 -16074.047,E2 -16074.047} C_VEL
LIN {X 0,Y 304.265,Z 436.244,A -85,B 0,C 180,E1 -16076.254,E2 -16076.254} C_VEL
LIN {X 0,Y 304.731,Z 431.9,A -85,B 0,C 180,E1 -16077.963,E2 -16077.963} C_VEL
LIN {X 0,Y 305.263,Z 426.726,A -85,B 0,C 180,E1 -16079.567,E2 -16079.567} C_VEL
LIN {X 0,Y 305.833,Z 421.739,A -85,B 0,C 180,E1 -16080.833,E2 -16080.833} C_VEL
LIN {X 0,Y 306.462,Z 415.548,A -85,B 0,C 180,E1 -16082.142,E2 -16082.142} C_VEL
LIN {X 0,Y 307.125,Z 408.974,A -85,B 0,C 180,E1 -16083.298,E2 -16083.298} C_VEL
LIN {X 0,Y 307.947,Z 400.647,A -85,B 0,C 180,E1 -16084.5,E2 -16084.5} C_VEL
LIN {X 0,Y 308.689,Z 391.195,A -85,B 0,C 180,E1 -16085.596,E2 -16085.596} C_VEL
LIN {X 0,Y 307.252,Z 381.088,A -85,B 0,C 180,E1 -16086.581,E2 -16086.581} C_VEL
LIN {X 0,Y 305.234,Z 370.628,A -85,B 0,C 180,E1 -16087.374,E2 -16087.374} C_VEL
LIN {X 0,Y 304.136,Z 364.94,A -85,B 0,C 180,E1 -16087.744,E2 -16087.744} C_VEL
LIN {X 0,Y 304.272,Z 361.402,A -85,B 0,C 180,E1 -16091.258,E2 -16091.258} C_VEL
LIN {X 0,Y 304.591,Z 357.008,A -85,B 0,C 180,E1 -16095.709,E2 -16095.709} C_VEL
LIN {X 0,Y 304.677,Z 356.092,A -85,B 0,C 180,E1 -16096.662,E2 -16096.662} C_VEL
LIN {X 0,Y 304.784,Z 355.333,A -85,B 0,C 180,E1 -16098.021,E2 -16098.021} C_VEL
LIN {X 0,Y 305.581,Z 355.233,A -85,B 0,C 180,E1 -16102.067,E2 -16102.067} C_VEL
LIN {X 0,Y 305.656,Z 355.223,A -85,B 0,C 180,E1 -16104.721,E2 -16104.721} C_VEL
LIN {X 0,Y 305.95,Z 355.186,A -85,B 0,C 180,E1 -16108.682,E2 -16108.682} C_VEL
LIN {X 0,Y 305.948,Z 355.185,A -85,B 0,C 180,E1 -16111.315,E2 -16111.315} C_VEL
LIN {X 0,Y 305.844,Z 355.198,A -85,B 0,C 180,E1 -16116.596,E2 -16116.596} C_VEL
LIN {X 0,Y 305.725,Z 355.213,A -85,B 0,C 180,E1 -16119.258,E2 -16119.258} C_VEL
LIN {X 0,Y 305.579,Z 355.231,A -85,B 0,C 180,E1 -16123.295,E2 -16123.295} C_VEL
LIN {X 0,Y 305.582,Z 355.233,A -85,B 0,C 180,E1 -16126.019,E2 -16126.019} C_VEL
LIN {X 0,Y 305.564,Z 355.235,A -85,B 0,C 180,E1 -16129.444,E2 -16129.444} C_VEL
LIN {X 0,Y 305.478,Z 355.244,A -85,B 0,C 180,E1 -16133.04,E2 -16133.04} C_VEL
LIN {X 0,Y 305.534,Z 355.236,A -85,B 0,C 180,E1 -16136.226,E2 -16136.226} C_VEL
LIN {X 0,Y 305.482,Z 355.244,A -85,B 0,C 180,E1 -16139.049,E2 -16139.049} C_VEL
LIN {X 0,Y 305.451,Z 355.25,A -85,B 0,C 180,E1 -16143.516,E2 -16143.516} C_VEL
LIN {X 0,Y 305.49,Z 355.242,A -85,B 0,C 180,E1 -16146.735,E2 -16146.735} C_VEL
LIN {X 0,Y 305.482,Z 355.244,A -85,B 0,C 180,E1 -16150.608,E2 -16150.608} C_VEL
LIN {X 0,Y 305.53,Z 355.237,A -85,B 0,C 180,E1 -16154.516,E2 -16154.516} C_VEL
LIN {X 0,Y 305.488,Z 355.242,A -85,B 0,C 180,E1 -16158.153,E2 -16158.153} C_VEL
LIN {X 0,Y 305.506,Z 355.24,A -85,B 0,C 180,E1 -16161.604,E2 -16161.604} C_VEL
LIN {X 0,Y 305.449,Z 355.251,A -85,B 0,C 180,E1 -16164.887,E2 -16164.887} C_VEL
LIN {X 0,Y 305.438,Z 355.25,A -85,B 0,C 180,E1 -16168.355,E2 -16168.355} C_VEL
LIN {X 0,Y 305.507,Z 355.24,A -85,B 0,C 180,E1 -16171.114,E2 -16171.114} C_VEL
LIN {X 0,Y 305.56,Z 355.234,A -85,B 0,C 180,E1 -16174.089,E2 -16174.089} C_VEL
LIN {X 0,Y 305.542,Z 355.24,A -85,B 0,C 180,E1 -16178.408,E2 -16178.408} C_VEL
LIN {X 0,Y 305.588,Z 355.229,A -85,B 0,C 180,E1 -16181.219,E2 -16181.219} C_VEL
LIN {X 0,Y 305.636,Z 355.223,A -85,B 0,C 180,E1 -16185.35,E2 -16185.35} C_VEL
LIN {X 0,Y 305.628,Z 355.224,A -85,B 0,C 180,E1 -16189.401,E2 -16189.401} C_VEL
LIN {X 0,Y 305.783,Z 355.206,A -85,B 0,C 180,E1 -16191.579,E2 -16191.579} C_VEL
LIN {X 0,Y 305.138,Z 355.291,A -85,B 0,C 180,E1 -16192.677,E2 -16192.677} C_VEL
LIN {X 0,Y 302.316,Z 355.646,A -85,B 0,C 180,E1 -16194.463,E2 -16194.463} C_VEL
LIN {X 0,Y 299.921,Z 355.942,A -85,B 0,C 180,E1 -16195.913,E2 -16195.913} C_VEL
LIN {X 0,Y 298.904,Z 356.063,A -85,B 0,C 180,E1 -16197.035,E2 -16197.035} C_VEL
LIN {X 0,Y 298.828,Z 356.071,A -85,B 0,C 180,E1 -16197.415,E2 -16197.415} C_VEL
LIN {X 0,Y 298.999,Z 356.055,A -85,B 0,C 180,E1 -16200.001,E2 -16200.001} C_VEL
LIN {X 0,Y 298.829,Z 356.071,A -85,B 0,C 180,E1 -16202.697,E2 -16202.697} C_VEL
LIN {X 0,Y 298.788,Z 356.076,A -85,B 0,C 180,E1 -16206.755,E2 -16206.755} C_VEL
LIN {X 0,Y 298.671,Z 356.094,A -85,B 0,C 180,E1 -16209.482,E2 -16209.482} C_VEL
LIN {X 0,Y 298.544,Z 356.111,A -85,B 0,C 180,E1 -16213.617,E2 -16213.617} C_VEL
LIN {X 0,Y 298.54,Z 356.107,A -85,B 0,C 180,E1 -16216.41,E2 -16216.41} C_VEL
LIN {X 0,Y 298.503,Z 356.115,A -85,B 0,C 180,E1 -16219.656,E2 -16219.656} C_VEL
LIN {X 0,Y 298.45,Z 356.122,A -85,B 0,C 180,E1 -16223.599,E2 -16223.599} C_VEL
LIN {X 0,Y 298.482,Z 356.115,A -85,B 0,C 180,E1 -16226.576,E2 -16226.576} C_VEL
LIN {X 0,Y 298.414,Z 356.124,A -85,B 0,C 180,E1 -16229.643,E2 -16229.643} C_VEL
LIN {X 0,Y 298.389,Z 356.128,A -85,B 0,C 180,E1 -16232.802,E2 -16232.802} C_VEL
LIN {X 0,Y 298.438,Z 356.123,A -85,B 0,C 180,E1 -16236.809,E2 -16236.809} C_VEL
LIN {X 0,Y 298.383,Z 356.131,A -85,B 0,C 180,E1 -16241.09,E2 -16241.09} C_VEL
LIN {X 0,Y 298.384,Z 356.13,A -85,B 0,C 180,E1 -16245.044,E2 -16245.044} C_VEL
LIN {X 0,Y 298.458,Z 356.26,A -85,B 0,C 180,E1 -16248.898,E2 -16248.898} C_VEL
LIN {X 0,Y 299.491,Z 361.694,A -85,B 0,C 180,E1 -16252.927,E2 -16252.927} C_VEL
LIN {X 0,Y 300.014,Z 365.768,A -85,B 0,C 180,E1 -16255.793,E2 -16255.793} C_VEL
LIN {X 0,Y 299.865,Z 368.384,A -85,B 0,C 180,E1 -16257.538,E2 -16257.538} C_VEL
LIN {X 0,Y 299.021,Z 374.017,A -85,B 0,C 180,E1 -16261.198,E2 -16261.198} C_VEL
LIN {X 0,Y 298.07,Z 381.035,A -85,B 0,C 180,E1 -16265.633,E2 -16265.633} C_VEL
LIN {X 0,Y 297.512,Z 386.852,A -85,B 0,C 180,E1 -16269.249,E2 -16269.249} C_VEL
LIN {X 0,Y 297.159,Z 391.383,A -85,B 0,C 180,E1 -16271.916,E2 -16271.916} C_VEL
LIN {X 0,Y 298.56,Z 403.311,A -85,B 0,C 180,E1 -16272.625,E2 -16272.625} C_VEL
LIN {X 0,Y 299.504,Z 413.453,A -85,B 0,C 180,E1 -16273.472,E2 -16273.472} C_VEL
LIN {X 0,Y 300.029,Z 422.297,A -85,B 0,C 180,E1 -16274.399,E2 -16274.399} C_VEL
LIN {X 0,Y 300.175,Z 429.103,A -85,B 0,C 180,E1 -16275.251,E2 -16275.251} C_VEL
LIN {X 0,Y 299.297,Z 437.038,A -85,B 0,C 180,E1 -16276.421,E2 -16276.421} C_VEL
LIN {X 0,Y 298.699,Z 442.77,A -85,B 0,C 180,E1 -16277.431,E2 -16277.431} C_VEL
LIN {X 0,Y 298.006,Z 449.176,A -85,B 0,C 180,E1 -16278.783,E2 -16278.783} C_VEL
LIN {X 0,Y 297.398,Z 455.687,A -85,B 0,C 180,E1 -16280.48,E2 -16280.48} C_VEL
LIN {X 0,Y 297.039,Z 459.912,A -85,B 0,C 180,E1 -16281.84,E2 -16281.84} C_VEL
LIN {X 0,Y 296.766,Z 463.403,A -85,B 0,C 180,E1 -16283.201,E2 -16283.201} C_VEL
LIN {X 0,Y 296.642,Z 466.254,A -85,B 0,C 180,E1 -16284.564,E2 -16284.564} C_VEL
LIN {X 0,Y 296.666,Z 468.516,A -85,B 0,C 180,E1 -16285.926,E2 -16285.926} C_VEL
LIN {X 0,Y 296.619,Z 470.132,A -85,B 0,C 180,E1 -16287.286,E2 -16287.286} C_VEL
LIN {X 0,Y 296.615,Z 471.195,A -85,B 0,C 180,E1 -16288.644,E2 -16288.644} C_VEL
LIN {X 0,Y 296.672,Z 471.775,A -85,B 0,C 180,E1 -16290.002,E2 -16290.002} C_VEL
LIN {X 0,Y 296.598,Z 471.876,A -85,B 0,C 180,E1 -16291.36,E2 -16291.36} C_VEL
LIN {X 0,Y 296.593,Z 471.474,A -85,B 0,C 180,E1 -16292.718,E2 -16292.718} C_VEL
LIN {X 0,Y 296.608,Z 470.475,A -85,B 0,C 180,E1 -16294.078,E2 -16294.078} C_VEL
LIN {X 0,Y 296.627,Z 468.701,A -85,B 0,C 180,E1 -16295.662,E2 -16295.662} C_VEL
